//模具切刀
fbMouldCam(
	Reset:=stSysState.bReset , 
	bCamInExecute:=stMouldCam.bCamInExecute , 
	bCreatTable:=stMouldCam.bCreatTable , 
	iTable:=TableNo.Mould , 
	iTableSel:= , 
	fEnterPos:=arrAxisPar[AxisNo.Mould].arrTargetPoint[2] , 
	fLeavePos:=arrAxisPar[AxisNo.Mould].arrTargetPoint[1] , 
	fMainPos:=ProductPar.parPublic.fMainPos , 
	axisSlave:=arrAxis[AxisNo.Mould] , 
	axisMaster:=arrAxis[VirAxisNo.VirMain] , 
	bCreatTableDone=>stMouldCam.bCreatTableDone , 
	bCreatTableError=>stMouldCam.bCreatTableError , 
	bError=>stMouldCam.bError , 
	bReady=>stMouldCam.bReady , 
	bInSync=>stMouldCam.bInSync );
	
//裁切切刀
fbCuterCam(
	Reset:=stSysState.bReset , 
	bCamInExecute:=stCuterCam.bCamInExecute , 
	bCreatTable:=stCuterCam.bCreatTable , 
	iTable:=TableNo.Cuter , 
	iTableSel:= ,
	fEnterPos:=arrAxisPar[AxisNo.Cuter].arrTargetPoint[2] , //裁切切入点角度
	fLeavePos:=arrAxisPar[AxisNo.Cuter].arrTargetPoint[1] , //裁切切尽点角度
	fMainPos:=ProductPar.parPublic.fMainPos , 
	axisSlave:=arrAxis[AxisNo.Cuter] , 
	axisMaster:=arrAxis[VirAxisNo.VirMain] , 
	bCreatTableDone=>stCuterCam.bCreatTableDone , 
	bCreatTableError=>stCuterCam.bCreatTableError , 
	bError=>stCuterCam.bError , 
	bReady=>stCuterCam.bReady , 
	bInSync=>stCuterCam.bInSync );

//CCD压片升降
fbCCDPressCam(
	Reset:=stSysState.bReset , 
	bCamInExecute:=stCCDPressCam.bCamInExecute , 
	bCreatTable:=stCCDPressCam.bCreatTable , 
	iTable:=TableNo.CCDPress , 
	fMainPos:=ProductPar.parPublic.fMainPos , 
	fPressPos:=arrAxisPar[AxisNo.CCDPressPush].arrTargetPoint[2]  , 
	fLeavePos:=arrAxisPar[AxisNo.CCDPressPush].arrTargetPoint[1] , 
	axisSlave:=arrAxis[AxisNo.CCDPressPush]  , 
	axisMaster:=arrAxis[VirAxisNo.VirMain]  , 
	bCreatTableDone=>stCCDPressCam.bCreatTableDone , 
	bCreatTableError=>stCCDPressCam.bCreatTableError , 
	bError=>stCCDPressCam.bError , 
	bReady=>stCCDPressCam.bReady , 
	bInSync=>stCCDPressCam.bInSync );
	
//皮带虚轴
fbVirBeltCam(
	Reset:=stSysState.bReset , 
	bCamInExecute:=stVirBeltCam.bCamInExecute , 
	bCreatTable:=stVirBeltCam.bCreatTable , 
	iTable:=TableNo.VirBelt , 
	fMainPos:=ProductPar.parPublic.fMainPos , 
	fBeltSpacePos:=PolePar.fBeltSpacePos , 
	axisSlave:=arrAxis[VirAxisNo.VirBelt]  , 
	axisMaster:=arrAxis[VirAxisNo.VirMain] , 
	bCreatTableDone=>stVirBeltCam.bCreatTableDone , 
	bCreatTableError=>stVirBeltCam.bCreatTableError , 
	bError=>stVirBeltCam.bError , 
	bReady=>stVirBeltCam.bReady , 
	bInSync=>stVirBeltCam.bInSync );
(*	
//NG踢料
fbNGPushCam(
	Reset:=stSysState.bReset , 
	bCamInExecute:=stNGPushCam.bCamInExecute , 
	bCreatTable:=stNGPushCam.bCreatTable , 
	iTable:=TableNo.NgPush , 
	iTableSel:= , 
	fEnterPos:=arrAxisPar[AxisNo.NGPush2].arrTargetPoint[2] , //NG打料预踢角度 , 
	fLeavePos:=arrAxisPar[AxisNo.NGPush2].arrTargetPoint[1] , //NG打料踢后角度 , 
	fMainPos:=ProductPar.parPublic.fMainPos , 
	axisSlave:=arrAxis[AxisNo.NGPush2] , 
	axisMaster:=arrAxis[VirAxisNo.VirMain] , 
	bCreatTableDone=>stNGPushCam.bCreatTableDone , 
	bCreatTableError=>stNGPushCam.bCreatTableError , 
	bError=>stNGPushCam.bError , 
	bReady=>stNGPushCam.bReady , 
	bInSync=>stNGPushCam.bInSync );
	*)
END_ACTION

ACTION F12TensionCall:


	fbPoleBufferTen.bTensionOK:=stUwindTen.bTensionOK;
	
	fbPoleBufferTen(
	bReset:=                               stSysState.bReset , 
	fAuxDriverDiameter:=            PolePar.Machine.fAuxDriverInDiameter ,  
	fDDRDiameter:=                    PolePar.Machine.fMQDriverDiameter ,  
	fPoleWith:=                           PolePar.fPoleWidth , 
    fCompensation:=                   fPoleBufferCompensation , 
    fDanceBlancePos:=                arrAxisPar[AxisNo.BuffeLine].arrTargetPoint[1] ,  
   	bPositiveLimit:=                     arrAxisCtrl[AxisNo.BuffeLine].Io.biPosLimit   , 
	bNegativeLimit:=                   arrAxisCtrl[AxisNo.BuffeLine].Io.biNegLimit      , 
	bTensionOK:=                       fbPoleBufferTen.bTensionOK     , 
	fMainVel:=                            PolePar.iMainVel         , 
	bReady=>                            stBufferTen.bReady , 
	bError=>                              stBufferTen.bError , 
	bInSync=>                            stBufferTen.bInSync, 
	VirMain:=                             arrAxis[VirAxisNo.VirMain], 
	//AuxDriver:=                          arrAxis[AxisNo.DriverAux] ,
	DDRDriver:=                         arrAxis[AxisNo.DriverDDR]  ,
	VirDriver:=                           arrAxis[VirAxisNo.VirDriver]  ,
	BufferLine:=                         arrAxis[AxisNo.BuffeLine] ,  
	bTenExecute:=                     stBufferTen.bExecute   );
	
	//放卷张力
PolePar.MQ.TenCcw_WindL:=PolePar.MQ.TenCcw_WindR:=FALSE;
	fbUwindTen(
		bReset:=stSysState.bReset , 
		bCcwL:=PolePar.MQ.TenCcw_WindL, //左放卷方向
		bCcwR:=PolePar.MQ.TenCcw_WindR,//右放卷方向
		bWindSel:=PolePar.MQ.bWindSelect, //左右卷选择
		fDiaMin:=250,//最小卷径		
		fDiaMax:=800,//最大卷径
		//fDanserDegree:=arrAxisCtrl[AxisNo.PoleTension].Status.fActPos , 
		fActTorque:= SEL(iPartSelect=1   , iActDriveTorque[2],    iActDriveTorque[1] )    , 
		fSetTorque:= SEL(iPartSelect=1   , iTargetTorque[2],       iTargetTorque[1] )      , 
		PidSwitch:=PolePar.MQ.WindPidSwitch ,
		bTenExecute:=stUwindTen.bTenExecute , 
		bStudyExecute:=stUwindTen.bStudyExecute AND stUwindTen.fStudyDiameter>0, 
		fStudyDiameter:=stUwindTen.fStudyDiameter , 
		fDriveDiameter:=PolePar.Machine.fMQDriverDiameter, 
		fPoleWith:=PolePar.fPoleWidth , 
		fCompensation:= , 
		fDancerMinPos:=PolePar.MQ.AuxDriverTenMinPos,//摆杆最小角度
		fDancerMaxPos:=PolePar.MQ.AuxDriverTenMaxPos,//摆杆最大角度
		fDanceBlancePos:=PolePar.MQ.AuxDriverTenBlancePos , //摆杆平衡角度
		fDanserDegree:=stAuxDriverTen.fDanserDegree , //摆杆实时角度
		//fDancerMinPos:=PolePar.MQ.WindTenMinPos , 
		//fDancerMaxPos:=PolePar.MQ.WindTenMaxPos , 
		//fDanceBlancePos:=PolePar.MQ.WindTenBlancePos , 
		bReady=>stUwindTen.bReady , 
		bTensionOK=>stUwindTen.bTensionOK , 
		bError=>stUwindTen.bError , 
		fWindDiameterTemp=>stUwindTen.fWindDiameter,
		VirMain:=arrAxis[VirAxisNo.VirMain] , 
		Master:=arrAxis[VirAxisNo.VirDriver] , 
		SlaveL:=arrAxis[AxisNo.UnWind_L], 
		SlaveR:=arrAxis[AxisNo.UnWind_R], 
		Driver:=arrAxis[AxisNo.DriverDDR] , 
		TimerAxis:=arrAxis[NameNo.VirTimeWind] , 
		TensionAxis:=arrAxis[AxisNo.PoleTension] , 
		Table:=PolePar.MQ.WindTenTable ,
		AxisNoBuffeLine :=AxisNo.BuffeLine);
	

		
		
(*
//左放卷张力

fbUwindLTen(
	bReset:=stSysState.bReset , 
	bCcw:=PolePar.MQ.TenCcw_WindL , 
	fDanserDegree:=stUwindLTen.fDanserDegree , 
	//fWindDiameter:=stUwindLTen.fWindDiameter  , 
	fActTorque:= SEL(iPartSelect=1   , iActDriveTorque[2],    iActDriveTorque[1] )    , 
	fSetTorque:= SEL(iPartSelect=1   , iTargetTorque[2],       iTargetTorque[1] )      , 
	PidSwitch:=TRUE , //PolePar.MQ.WindPidSwitch
	bTenExecute:=stUwindLTen.bTenExecute , 
	bStudyExecute:=stUwindLTen.bStudyExecute , 
	fStudyDiameter:=stUwindLTen.fStudyDiameter , 
	fDriveDiameter:=PolePar.Machine.fAuxDriverInDiameter , 
	fPoleWith:=PolePar.fPoleWidth , 
	fCompensation:= , 
	fDancerMinPos:=PolePar.MQ.WindTenMinPos , 
	fDancerMaxPos:=PolePar.MQ.WindTenMaxPos , 
	fDanceBlancePos:=PolePar.MQ.WindTenBlancePos , 
	bReady=>stUwindLTen.bReady , 
	bTensionOK=>stUwindLTen.bTensionOK , 
	bError=>stUwindLTen.bError , 
	VirMain:=arrAxis[VirAxisNo.VirMain] , 
	Master:=arrAxis[VirAxisNo.VirDriver] , 
	Slave:=arrAxis[AxisNo.UnWind_L] , 
	Driver:=arrAxis[AxisNo.DriverAux] , 
	TimerAxis:=arrAxis[NameNo.VirTimeWind] , 
	TensionAxis:=arrAxis[AxisNo.PoleTension] , 
	Table:=PolePar.MQ.WindTenTable );
	stUwindLTen.fDanserDegree:=arrAxisCtrl[AxisNo.PoleTension].Status.fActPos;
	PolePar.MQ.TenCcw_WindL:=FALSE;
	
	stUwindLTen.fWindDiameter  ;
	fbUwindLTen.fWindDiameter;
	fbUwindLTen.fDiameterCalculate;
	fbUwindLTen.fWindDiameterTemp;
	
//右放卷张力
fbUwindRTen(	
	bReset:=stSysState.bReset , 
	bCcw:=PolePar.MQ.TenCcw_WindR , 
	fDanserDegree:=stUwindRTen.fDanserDegree , 
	//fWindDiameter:=stUwindRTen.fWindDiameter , 
	fActTorque:= SEL(iPartSelect=1   , iActDriveTorque[2],    iActDriveTorque[1] )    , 
	fSetTorque:= SEL(iPartSelect=1   , iTargetTorque[2],       iTargetTorque[1] )      , 
	PidSwitch:=TRUE, //PolePar.MQ.WindPidSwitch 
	bTenExecute:=stUwindRTen.bTenExecute , 
	bStudyExecute:=stUwindRTen.bStudyExecute , 
	fStudyDiameter:=stUwindRTen.fStudyDiameter , 
	fDriveDiameter:=PolePar.Machine.fAuxDriverInDiameter , 
	fPoleWith:=PolePar.fPoleWidth , 
	fCompensation:= ,
	fDancerMinPos:=PolePar.MQ.WindTenMinPos , 
	fDancerMaxPos:=PolePar.MQ.WindTenMaxPos , 
	fDanceBlancePos:=PolePar.MQ.WindTenBlancePos , 
	bReady=>stUwindRTen.bReady , 
	bTensionOK=>stUwindRTen.bTensionOK , 
	bError=>stUwindRTen.bError , 
	VirMain:=arrAxis[VirAxisNo.VirMain] , 
	Master:=arrAxis[VirAxisNo.VirDriver] , 
	Slave:=arrAxis[AxisNo.UnWind_R]  , 
	Driver:=arrAxis[AxisNo.DriverAux] , 
	TimerAxis:=arrAxis[NameNo.VirTimeWind], 
	TensionAxis:=arrAxis[AxisNo.PoleTension] , 
	Table:=PolePar.MQ.WindTenTable );
	
	
	
	stUwindRTen.fDanserDegree:=arrAxisCtrl[AxisNo.PoleTension].Status.fActPos;
	PolePar.MQ.TenCcw_WindR:=FALSE;
	
	stUwindRTen.fWindDiameter  ;
	fbUwindRTen.fWindDiameter;
	fbUwindRTen.fDiameterCalculate;
	fbUwindRTen.fWindDiameterTemp;
*)	
//辅驱张力
stAuxDriverTen.fWindDiameter:=stAuxDriverTen.fStudyDiameter:=PolePar.Machine.fAuxDriverInDiameter;
PolePar.MQ.TenCcw_AuxDriver:=FALSE;
fbAuxDriverTen(
	bReset:=stSysState.bReset , 
	bCcw:=PolePar.MQ.TenCcw_AuxDriver , 
	fDanserDegree:=stAuxDriverTen.fDanserDegree , 
	fWindDiameter:=stAuxDriverTen.fWindDiameter , 
	PidSwitch:=FALSE , //PolePar.MQ.AuxDriverPidSwitch
	bTenExecute:=stAuxDriverTen.bTenExecute , 
	bStudyExecute:=FALSE, //stAuxDriverTen.bStudyExecute
	fStudyDiameter:=stAuxDriverTen.fStudyDiameter , 
	fPoleWith:=PolePar.fPoleWidth , 
	fCompensation:= , 
	fDancerMinPos:=PolePar.MQ.AuxDriverTenMinPos , 
	fDancerMaxPos:=PolePar.MQ.AuxDriverTenMaxPos , 
	fDanceBlancePos:=PolePar.MQ.AuxDriverTenBlancePos , 
	bReady=>stAuxDriverTen.bReady , 
	bTensionOK=>stAuxDriverTen.bTensionOK , 
	bError=>stAuxDriverTen.bError , 
	VirMain:=arrAxis[VirAxisNo.VirMain] , 
	Master:=arrAxis[VirAxisNo.VirDriver] , 
	Slave:=arrAxis[AxisNo.DriverAux] , 
	TimerAxis:=arrAxis[NameNo.VirTimeWind] , 
	Table:=PolePar.MQ.AuxDriverTenTable );
END_ACTION

ACTION F13ClearBelt:
//一键皮带清料
rtClearBelt[1](CLK:=SysPart.hmiClearBelt , Q=> );
rtClearBelt[2](CLK:= , Q=> );
rtClearBelt[3](CLK:= , Q=> );
rtClearBelt[4](CLK:= , Q=> );
rtClearBelt[5](CLK:= , Q=> );
tonClearBelt[1](In:=,PT:=T#200MS);
tonClearBelt[2](In:=,PT:=T#200MS);
tonClearBelt[3](In:=,PT:=T#200MS);
tonClearBelt[4](In:=,PT:=T#200MS);	
tonClearBelt[5](In:=,PT:=T#200MS);	
tonClearBelt[6](In:=,PT:=T#200MS);	
tonClearBelt[7](In:=,PT:=T#200MS);
tonClearBelt[8](In:=,PT:=T#200MS);
tonClearBelt[9](In:=,PT:=T#200MS);
tonClearBelt[10](In:=,PT:=T#200MS);
IF rtClearBelt[1].Q THEN
	iClearBeltStep:=88;//皮带清料触发
END_IF;

CASE iClearBeltStep OF
///////////////////////////////////////////////////////////凸轮耦合/////////////////////////////////////////////////////
88://有关气缸动作
	arrCyCtrl[CYNo.NGRevBeltTension].Cmd.bON:=TRUE;
	arrCyCtrl[CYNo.NGRevBeltUpDown].Cmd.bON:=TRUE;
	arrCyCtrl[CYNo.DustRevBeltUpDown].Cmd.bON:=TRUE;
	IF	arrCyCtrl[CyNo.NGRevBeltUpDown].Status.ONState AND arrCyCtrl[CYNo.DustRevBeltUpDown].Status.ONState THEN
		iClearBeltStep:=90;//		
	END_IF
	
90://凸轮/张力解耦
	bMethodTenBufferDisEnable:=TRUE;
	bMethodCamDisEnable:=TRUE;
	iClearBeltStep:=100;//	
	
100://判断是否解耦完成
	IF NOT bMethodTenBufferDisEnable AND NOT bMethodCamDisEnable THEN
		iClearBeltStep:=110;
	END_IF
110://主轴清0
	IF arrAxisCtrl[VirAxisNo.VirMain].Status.fModuloActPos<>0 THEN
		arrAxisCtrl[VirAxisNo.VirMain].Cmd.fSetPos:=arrAxisCtrl[VirAxisNo.VirMain].Status.fActPos-arrAxisCtrl[VirAxisNo.VirMain].Status.fModuloActPos+360;
		arrAxisCtrl[VirAxisNo.VirMain].Cmd.bSetPos:=TRUE;
	END_IF
	iClearBeltStep:=120;
120://皮带虚轴耦合
	IF NOT stVirBeltCam.bInSync THEN
		stVirBeltCam.bCamInExecute:=TRUE;
	ELSE
		iClearBeltStep:=130;
	END_IF	
130://皮带齿合
	IF NOT stCuterBeltGear.bInGear THEN
		stCuterBeltGear.bEnable:=TRUE;
	END_IF	
	IF NOT stNGReverseBeltGear.bInGear THEN
		stNGReverseBeltGear.bEnable:=TRUE;
	END_IF		
	IF NOT stDedustBeltGear.bInGear THEN
		stDedustBeltGear.bEnable:=TRUE;
	END_IF
	IF NOT stDedustReverseBeltGear.bInGear THEN
		stDedustReverseBeltGear.bEnable:=TRUE;
	END_IF

	IF NOT stSubBelt1Gear.bInGear THEN
		stSubBelt1Gear.bEnable:=TRUE;
	END_IF

	IF NOT stSubBelt2Gear.bInGear THEN
		bSubBelt2fratio:=TRUE;
		stSubBelt2Gear.bEnable:=TRUE;
	END_IF	
	
	IF NOT stSubBelt3Gear.bInGear THEN
		bSubBelt3fratio:=TRUE;
		stSubBelt3Gear.bEnable:=TRUE;
	END_IF		

	IF stCuterBeltGear.bInGear AND stNGReverseBeltGear.bInGear AND stDedustBeltGear.bInGear AND stDedustReverseBeltGear.bInGear AND 
	     stSubBelt1Gear.bInGear AND  stSubBelt2Gear.bInGear AND  stSubBelt3Gear.bInGear THEN
    	iClearBeltStep:=140;		
	END_IF
140://主轴运动40个周期
	arrAxisCtrl[VirAxisNo.VirMain].Cmd.bDynamitcsParSel:=1;
	arrAxisCtrl[VirAxisNo.VirMain].Cmd.fPositon_of_Abs:=arrAxisCtrl[VirAxisNo.VirMain].Status.fActPos-arrAxisCtrl[VirAxisNo.VirMain].Status.fModuloActPos+40*360;
	arrAxisPar[VirAxisNo.VirMain].fVelocity_of_Abs:=PolePar.iMainVel*6;
	arrAxisCtrl[VirAxisNo.VirMain].Cmd.bMoveAbs:=TRUE;
	IF arrAxisCtrl[VirAxisNo.VirMain].Status.Moving THEN
		iClearBeltStep:=150;
	END_IF
150://判断主轴运动完成
	IF arrAxisCtrl[VirAxisNo.VirMain].Status.NoMoving AND NOT arrAxisCtrl[VirAxisNo.VirMain].Cmd.bMoveAbs THEN
		iClearBeltStep:=160;
	END_IF
160://清除皮带记忆
	MEMSET(ADR(BeltData),0,SIZEOF(BeltData));
	iClearBeltStep:=170;
170://
	SysPart.hmiClearBelt:=FALSE;
	iClearBeltStep:=666;

END_CASE
END_ACTION

ACTION Product:

//切刀计数
rtCount2(CLK:=arrAxisCtrl[VirAxisNo.VirMain].Status.fModuloActPos>=10 AND arrAxisCtrl[VirAxisNo.VirMain].Status.fModuloActPos<=100);
IF rtCount2.Q THEN
	Production.OutFlag1:=TRUE;//产能计数
END_IF

////////////////////////////////////////////////////////////////NG剔废////////// NG分类 //////////////////////////////////////////////////////
ProductPar.iModeEN.bNG1PushEN:=ProductPar.iModeEN.bNG2PushEN;
CASE iNGStep OF 
10://判断NG1&NG2是否动作 主轴静止或运行中
	IF (  NOT ProductPar.iModeEN.bEmptyRunEN AND NOT ProductPar.iModeEN.bSizeCCDEN AND BeltData[BeltNo.NGBox1+2].fPoleNGSizeNo<>30 ) THEN//BeltData[BeltNo.NGBox].iPanoramaNG<>1
		 iNGStep:=200;
	ELSIF  BeltData[BeltNo.NGBox1+2].fPoleNGSacnNo<>30   AND NOT ProductPar.iModeEN.bLineScanCCDEN  THEN //XianSaong_Up[2]<>30 OR XianSaong_Down[0]<>30  
		iNGStep:=300;
	ELSIF  BeltData[BeltNo.NGBox1+2].bYellowMark    OR  BeltData[BeltNo.NGBox1+2].bBlueMark  THEN//黄标
		iNGStep:=300;
	ELSE
		nInt[3]:=0;
		arrCyCtrl[EvNo.	NGPushInsideAir	].Cmd.bON:=FALSE;//踢NG料打开
		arrCyCtrl[EvNo.	NGPushInsideAir	].Cmd.bOFF:=TRUE;//踢NG料关闭		
		arrCyCtrl[EVNo.NGPushInsideVacuo].Cmd.bON:=TRUE;//踢NG料真空打开
		arrCyCtrl[EVNo.NGPushInsideVacuo].Cmd.bOFF:=FALSE;//踢NG料真空关闭		
		iNGStep:=666;
	END_IF

200:
	IF  NOT ProductPar.iModeEN.bEmptyRunEN   THEN//AND NOT  ProductPar.iModeEN.bP2PartEN
			IF REAL_TO_INT(BeltData[BeltNo.NGBox1+2].fPoleNGSizeNo)=1 THEN
				Production.NGFlag[49]:=TRUE;//尺寸总不良
				Production.NGFlag[1]:=TRUE;//极片长度不良
			ELSIF REAL_TO_INT(BeltData[BeltNo.NGBox1+2].fPoleNGSizeNo)=2 THEN
				Production.NGFlag[49]:=TRUE;//尺寸总不良
				Production.NGFlag[2]:=TRUE;//极片CIL宽度不良
			ELSIF REAL_TO_INT(BeltData[BeltNo.NGBox1+2].fPoleNGSizeNo)=3 THEN
				Production.NGFlag[49]:=TRUE;//尺寸总不良
				Production.NGFlag[3]:=TRUE;//极片宽度不良标志位
			ELSIF REAL_TO_INT(BeltData[BeltNo.NGBox1+2].fPoleNGSizeNo)=4 THEN
				Production.NGFlag[49]:=TRUE;//尺寸总不良
				Production.NGFlag[4]:=TRUE;//极耳宽度不良
			ELSIF REAL_TO_INT(BeltData[BeltNo.NGBox1+2].fPoleNGSizeNo)=5 THEN
				Production.NGFlag[49]:=TRUE;//尺寸总不良
				Production.NGFlag[5]:=TRUE;//极耳高度不良
			ELSIF REAL_TO_INT(BeltData[BeltNo.NGBox1+2].fPoleNGSizeNo)=6 THEN
				Production.NGFlag[49]:=TRUE;//尺寸总不良
				Production.NGFlag[6]:=TRUE;//极耳侧边距不良
			ELSIF REAL_TO_INT(BeltData[BeltNo.NGBox1+2].fPoleNGSizeNo)=7 THEN
				Production.NGFlag[49]:=TRUE;//尺寸总不良
				Production.NGFlag[7]:=TRUE;//极耳面积不良
			ELSIF REAL_TO_INT(BeltData[BeltNo.NGBox1+2].fPoleNGSizeNo)=8 THEN
				Production.NGFlag[49]:=TRUE;//尺寸总不良
				Production.NGFlag[8]:=TRUE;//圆角深度不良
			ELSIF REAL_TO_INT(BeltData[BeltNo.NGBox1+2].fPoleNGSizeNo)=9 THEN
				Production.NGFlag[49]:=TRUE;//尺寸总不良
				Production.NGFlag[9]:=TRUE;//极耳边缘角度不良
			ELSIF REAL_TO_INT(BeltData[BeltNo.NGBox1+2].fPoleNGSizeNo)=10 THEN
				Production.NGFlag[49]:=TRUE;//尺寸总不良
				Production.NGFlag[10]:=TRUE;//圆角宽度不良
			ELSIF REAL_TO_INT(BeltData[BeltNo.NGBox1+2].fPoleNGSizeNo)=11 THEN
				Production.NGFlag[49]:=TRUE;//尺寸总不良
				Production.NGFlag[11]:=TRUE;//圆角轮廓不良	
			ELSIF REAL_TO_INT(BeltData[BeltNo.NGBox1+2].fPoleNGSizeNo)=12 THEN
				Production.NGFlag[49]:=TRUE;//尺寸总不良
				Production.NGFlag[12]:=TRUE;//圆角面积不良		
			ELSIF REAL_TO_INT(BeltData[BeltNo.NGBox1+2].fPoleNGSizeNo)=13 THEN
				Production.NGFlag[49]:=TRUE;//尺寸总不良
				Production.NGFlag[13]:=TRUE;//圆角余料不良		
			ELSIF (BeltData[BeltNo.NGBox1+2].fPoleNGSizeNo<>1 AND BeltData[BeltNo.NGBox1+2].fPoleNGSizeNo<>2 AND BeltData[BeltNo.NGBox1+2].fPoleNGSizeNo<>3
				AND BeltData[BeltNo.NGBox1+2].fPoleNGSizeNo<>4 AND BeltData[BeltNo.NGBox1+2].fPoleNGSizeNo<>5 AND BeltData[BeltNo.NGBox1+2].fPoleNGSizeNo<>6
				 AND BeltData[BeltNo.NGBox1+2].fPoleNGSizeNo<>7  AND BeltData[BeltNo.NGBox1+2].fPoleNGSizeNo<>8  AND BeltData[BeltNo.NGBox1+2].fPoleNGSizeNo<>9
				 AND BeltData[BeltNo.NGBox1+2].fPoleNGSizeNo<>11  AND BeltData[BeltNo.NGBox1+2].fPoleNGSizeNo<>12  AND BeltData[BeltNo.NGBox1+2].fPoleNGSizeNo<>13
				) OR  BeltData[BeltNo.NGBox1+2].fPoleNGSizeNo=33  THEN  //尺寸检测其他不良 ,,,CCD超时
				Production.NGFlag[49]:=TRUE;//尺寸检测其他不良 ,,,CCD超时
				Production.NGFlag[14]:=TRUE;
			END_IF
	END_IF
		FOR i:=1 TO 20 DO
			IF i<20 THEN
				XianSaong[21-i]:=XianSaong[20-i];
				XianSaong1[21-i]:=XianSaong1[20-i];
			ELSE
				XianSaong[1]:=BeltData[BeltNo.NGBox1].iPanoramaNG;
				XianSaong1[1]:=REAL_TO_INT(BeltData[BeltNo.NGBox1].fPoleNGSizeNo);
			END_IF
		END_FOR
		iNGStep:=400;
300:
	 IF NOT ProductPar.iModeEN.bEmptyRunEN  THEN//AND NOT  ProductPar.iModeEN.bP2PartEN
			IF BeltData[BeltNo.NGBox1+2].fPoleNGSacnNo=1 THEN
				Production.NGFlag[48]:=TRUE;//线扫总不良
				Production.NGFlag[21]:=TRUE;//抓边失败
			ELSIF BeltData[BeltNo.NGBox1+2].fPoleNGSacnNo=2 THEN
				Production.NGFlag[48]:=TRUE;//线扫总不良
				Production.NGFlag[22]:=TRUE;//直边不良标志位
			ELSIF BeltData[BeltNo.NGBox1+2].fPoleNGSacnNo=3 THEN
				Production.NGFlag[48]:=TRUE;//线扫总不良
				Production.NGFlag[23]:=TRUE;//极片缺失
			ELSIF BeltData[BeltNo.NGBox1+2].fPoleNGSacnNo=4 THEN
				Production.NGFlag[48]:=TRUE;//线扫总不良
				Production.NGFlag[24]:=TRUE;//接带
			ELSIF BeltData[BeltNo.NGBox1+2].fPoleNGSacnNo=5 THEN
				Production.NGFlag[48]:=TRUE;//线扫总不良
				Production.NGFlag[25]:=TRUE;//线扫黄标
			ELSIF BeltData[BeltNo.NGBox1+2].fPoleNGSacnNo=6 THEN
				Production.NGFlag[48]:=TRUE;//线扫总不良
				Production.NGFlag[26]:=TRUE;//漏金属
			ELSIF BeltData[BeltNo.NGBox1+2].fPoleNGSacnNo=7 THEN
				Production.NGFlag[48]:=TRUE;//线扫总不良
				Production.NGFlag[27]:=TRUE;//气泡
			ELSIF BeltData[BeltNo.NGBox1+2].fPoleNGSacnNo=8 THEN
				Production.NGFlag[48]:=TRUE;//线扫总不良
				Production.NGFlag[28]:=TRUE;//暗条痕
			ELSIF BeltData[BeltNo.NGBox1+2].fPoleNGSacnNo=9 THEN
				Production.NGFlag[48]:=TRUE;//线扫总不良
				Production.NGFlag[29]:=TRUE;//亮条痕
			ELSIF BeltData[BeltNo.NGBox1+2].fPoleNGSacnNo=10 THEN
				Production.NGFlag[48]:=TRUE;//线扫总不良
				Production.NGFlag[30]:=TRUE;//破损
			ELSIF BeltData[BeltNo.NGBox1+2].fPoleNGSacnNo=11 THEN
				Production.NGFlag[48]:=TRUE;//线扫总不良
				Production.NGFlag[31]:=TRUE;//碎屑
			ELSIF BeltData[BeltNo.NGBox1+2].fPoleNGSacnNo=12 THEN
				Production.NGFlag[48]:=TRUE;//线扫总不良
				Production.NGFlag[33]:=TRUE;//脱碳
			ELSIF BeltData[BeltNo.NGBox1+2].fPoleNGSacnNo=29 THEN
				Production.NGFlag[48]:=TRUE;//线扫总不良
				Production.NGFlag[34]:=TRUE;//其他
			ELSIF BeltData[BeltNo.NGBox1+2].fPoleNGSacnNo=33 THEN
				Production.NGFlag[48]:=TRUE;//线扫总不良
				Production.NGFlag[32]:=TRUE;//通讯超时
(*			ELSIF BeltData[BeltNo.NGBox1+2].bYellowMark  THEN
				//Production.NGFlag[48]:=TRUE;//线扫总不良
				Production.NGFlag[33]:=TRUE;//感应器黄标*)
			END_IF
	END_IF
		iNGStep:=400;
400:
	arrCyCtrl[EvNo.	NGPushInsideAir	].Cmd.bON:=TRUE;//踢NG料破真空打开
	arrCyCtrl[EvNo.	NGPushInsideAir	].Cmd.bOFF:=FALSE;//踢NG料破真空关闭
	arrCyCtrl[EVNo.NGPushInsideVacuo].Cmd.bON:=FALSE;//踢NG料真空打开
	arrCyCtrl[EVNo.NGPushInsideVacuo].Cmd.bOFF:=TRUE;//踢NG料真空关闭
	BeltData[BeltNo.NGBox1+2].bHavePole:=FALSE;	
	BeltData[BeltNo.NGBox1+2].stPoleNo:='';
	nInt[3]:=1;		
	//BeltData[BeltNo.NGBox1].bHavePole:=FALSE;
	FOR i:=1 TO 50 DO//NG类型标志位复位
		Production.NGFlag[i]:=FALSE;
    	END_FOR
	iNGStep:=666;
END_CASE

IF iNGStep=300 THEN
	IF BeltData[BeltNo.NGBox1+1].bBlueMark OR BeltData[BeltNo.NGBox1+2].bBlueMark OR BeltData[BeltNo.NGBox1+3].bBlueMark THEN
		iNGState:=1;//接带踢废
	ELSIF BeltData[BeltNo.NGBox1+2].bYellowMark THEN
		IF BeltData[BeltNo.NGBox1+1].bYellowMark THEN
			iNGState:=2;//黄标跳切踢废
		ELSIF NOT BeltData[BeltNo.NGBox1+3].bYellowMark THEN
			iNGState:=3;//黄标单张踢废
		END_IF
	ELSIF BeltData[BeltNo.NGBox1+2].fPoleNGSacnNo=4 THEN
		iNGState:=4;//线扫接带
	ELSIF BeltData[BeltNo.NGBox1+2].fPoleNGSacnNo=5 THEN
		iNGState:=5;//线扫黄标
	END_IF
END_IF

aFB_ProductionDataLocal(
	NowTimeData:=System.StTime, (*当前系统时间*)
	OutFlag1:=Production.OutFlag1, (*产量计数标志1*)
	OutFlag2:=Production.OutFlag2, (*产量计数标志1*)
	NGFlag:=Production.NGFlag ,(*NG1计数标志*)(*扫码NG*)
	RunFlag:=stSysState.iMode=1,(*运行标志*)
	WaitFlag:=stSysState.iMode<>1 AND NOT stSysState.Alarming ,(*待料标志*)
	AlarmFlag:=stSysState.Alarming, (*故障标志*)
	DelDataAMBtn:= Production.HMI_DelDataAMBtn,(*白班数据清除按钮*)//HMI_DayCountZero
	DelDataPMBtn:= Production.HMI_DelDataPMBtn,(*夜班数据清除按钮*)//HMI_NightCountZero
	NowOutTotal=>Production.HMI_TotalCount ,(*当前班次加工总数*)
	NowRate=> Production.HMI_Qualified,(*当前班次良率*)
	NGClearAMBtn:=Production.HMI_NGClearAMBtn,//白班NG类型计数清零
	NGClearPMBtn:=Production.HMI_NGClearPMBtn,//夜班NG类型计数清零
	NowDay:= Production.SaveNowDay,(*数据移位时所保存当前日*)
	NowMonth:=Production.SaveNowMonth ,(*数据移位时所保存当前月*)
	DayHistory:= Production.DayReadDayHistory, (*历史日*)
	MonthHistory:= Production.DayReadMonthHistory,(*历史月*)
	TodayTotal:=Production.HMI_TodayTotal ,(*当天24H生产总数*)
	TodayOK:=Production.HMI_TodayOK , (*当天24H生产OK总数*)
	TodayNG:=Production.HMI_TodayNG , (*当天24H生产NG总数*)
	TodayTotal_AM:= Production.DayCountTotal,(*当天白班生产总数*)
	TodayTotal_PM:=Production.NightCountTotal,(*当天夜班生产总数*)
	TodayRate_AM:= Production.HMI_DayQualified,(*当天白班良率*)
	TodayRate_PM:=Production.HMI_NightQualified ,(*当天夜班良率*)
	OEE=> Production.HMI_OEE,//设备稼动率/稼动率
	TodayOK_AM:=Production.HMI_DayOkCount ,(*当天白班生产OK总数*)
	TodayOK_PM:= Production.HMI_NightOkCount,(*当天夜班生产OK总数*)
	TodayNG_AM:=Production.HMI_DayNgCount ,(*当天白班生产NG总数*)
	TodayNG_PM:=Production.HMI_NightNgCount , (*当天夜班生产NG总数*)
	TodayHour_AM:= Production.HourTimeDayCount,(*当天白班每小时产量ARRAY[8..19 ]*)
	TodayHour_PM:=Production.HourTimeNightCount ,(*当天夜班每小时产量ARRAY[0..23]*)
	TodayNGClass_AM:=Production.NgPerHourDayCount , (*当天白班各类NG数量ARRAY[1..30 ]*)
	TodayNGClass_PM:= Production.NgPerHourNightCount,(*当天夜班各类NG数量ARRAY[1..30 ]*)
	TodayRun_AM:= Production.DayRunTimeTotal,(*当天白班总运行时间合计/分*)
	TodayRun_PM:= Production.NightRunTimeTotal,(*当天夜班总运行时间合计/分*)
	TodayWait_AM:=Production.DayWaitTimeTotal , (*当天白班总待料时间合计/分*)
	TodayWait_PM:=Production.NightWaitTimeTotal , (*当天夜班总待料时间合计/分*)
	TodayAlarm_AM:=Production.DayAlarmTimeTotal ,(*当天白班总报警时间合计/分*)
	TodayAlarm_PM:=Production.NightAlarmTimeTotal, (*当天夜班总报警时间合计/分*)
	
	TodayRun_AMH:=Production.DayRunTime_min,(*当天白班每小时运行时间合计/分*)
	TodayRun_PMH:=Production.NightRunTime_min,(*当天夜班每小时运行时间合计/分*)
	TodayWait_AMH:=Production.DayWaitTime_min,(*当天白班每小时待料时间合计/分*)
	TodayWait_PMH:=Production.NightWaitTime_min,(*当天夜班每小时待料时间合计/分*)
	TodayAlarm_AMH:=Production.DayAlmTime_min,(*当天白班每小时报警时间合计/分*)
	TodayAlarm_PMH:=Production.NightAlmTime_min,(*当天夜班每小时报警时间合计/分*)
	
	HistoryRun_AMH:=Production.HisDayRunTime_min,(*历史每天白班每小时运行时间合计ARRAY[1..7 ]*)
	HistoryRun_PMH:=Production.HisNightRunTime_min,(*历史每天夜班每小时运行时间合计ARRAY[1..7 ]*)
	HistoryWait_AMH:=Production.HisDayWaitTime_min,(*历史每天白班每小时待料时间合计ARRAY[1..7 ]*)
	HistoryWait_PMH:=Production.HisNightWaitTime_min,(*历史每天夜班每小时待料时间合计ARRAY[1..7 ]*)
	HistoryAlarm_AMH:=Production.HisDayAlmTime_min,(*历史每天白班每小时报警时间合计ARRAY[1..7 ]*)
	HistoryAlarm_PMH:=Production.HisNightAlmTime_min,(*历史每天夜班每小时报警时间合计ARRAY[1..7 ]*)
	
	RunCnt_AM:=Production.nDayRunTimeCnt , (*白班运行时间计数*)
	RunCnt_PM:=Production.nNightRunTimeCnt ,(*夜班运行时间计数*)
	WaitCnt_AM:= Production.nDayWaitTimeCnt, (*白班待料时间计数*)
	WaitCnt_PM:=Production.nNightWaitTimeCnt ,(*夜班待料时间计数*)
	AlarmCnt_AM:=Production.nDayAlarmTimeCnt , (*白班报警时间计数*)
	AlarmCnt_PM:= Production.nNightAlarmTimeCnt,(*夜班报警时间计数*)
	
	HistoryTotal:=Production.HMI_HistoryTotal ,(*历史每天24H生产总数ARRAY[1..7 ]*)
	HistoryOK:=Production.HMI_HistoryOK ,(*历史每天24H生产OK总数ARRAY[1..7 ]*)
	HistoryNG:=Production.HMI_HistoryNG , (*历史每天24H生产NG总数ARRAY[1..7 ]*)
	HistoryTotal_AM:=Production.DayCountTotalHistory ,(*历史每天白班生产总数ARRAY[1..7 ]*)
	HistoryTotal_PM:=Production.NightCountTotalHistory ,(*历史每天夜班生产总数ARRAY[1..7 ]*)
	HistoryRate_AM:=Production.HMI_DayQualifiedHistory , (*历史每天白班良率ARRAY[1..7 ]*)
	HistoryRate_PM:=Production.HMI_NightQualifiedHistory,(*历史每天夜班良率ARRAY[1..7 ]*)
	HistoryOK_AM:=Production.HMI_DayOkCountHistory , (*历史每天白班生产OK总数ARRAY[1..7 ]*)
	HistoryOK_PM:=Production.HMI_NightOkCountHistory , (*历史每天夜班生产OK总数ARRAY[1..7 ]*)
	HistoryNG_AM:=Production.HMI_DayNgCountHistory ,(*历史每天白班生产NG总数ARRAY[1..7 ]*)
	HistoryNG_PM:= Production.HMI_NightNgCountHistory,(*历史每天夜班生产NG总数ARRAY[1..7 ]*)
	HistoryHour_AM:=Production.HourTimeDayCountHistory ,(*历史每天白班每小时产量ARRAY[1..7,8..19 ]*)
	HistoryHour_PM:=Production.HourTimeNightCountHistory ,(*历史每天夜班每小时产量ARRAY[1..7,0..23]*)
	HistoryNGClass_AM:= Production.NgPerHourDayCountHistory,(*历史每天白班各类NG数量ARRAY[1..7,1..30 ]*)
	HistoryNGClass_PM:= Production.NgPerHourNightCountHistory,(*历史每天夜班各类NG数量ARRAY[1..7,1..30 ]*)
	HistoryRun_AM:=Production.DayRunTimeTotalHistory , (*历史每天白班总运行时间合计ARRAY[1..7 ]*)
	HistoryRun_PM:= Production.NightRunTimeTotalHistory, (*历史每天夜班总运行时间合计ARRAY[1..7 ]*)
	HistoryWait_AM:= Production.DayWaitTimeTotalHistory,(*历史每天白班总待料时间合计ARRAY[1..7 ]*)
	HistoryWait_PM:= Production.NightWaitTimeTotalHistory, (*历史每天夜班总待料时间合计ARRAY[1..7 ]*)
	HistoryAlarm_AM:= Production.DayAlarmTimeTotalHistory,(*历史每天白班总报警时间合计ARRAY[1..7 ]*)
	HistoryAlarm_PM:= Production.NightAlarmTimeTotalHistory,(*历史每天夜班总报警时间合计ARRAY[1..7 ]*)

	TodayNgHour_Day:=Production.HMINgClassCount_Day,(*白班每种NG类型每小时统计 ,,,NG类型，小时*)
	TodayNgHour_Night:=Production.HMINgClassCount_Night,(*夜班每种NG类型每小时统计 ,,,NG类型，小时*)
	HisTodayNgHour_Day:=Production.HisHMINgClassCount_Day,//l历史白班每小时NG类型统计,,
	HisTodayNgHour_Night:=Production.HisHMINgClassCount_Night,//历史夜班每小时NG类型统计,,
		
	TodayNGQualified:=Production.HMI_TodayNGQualified,//当天白班各种NG类型NG率
	NightNGQualified:=Production.HMI_NightNGQualified,//当天夜班各种NG类型NG率	
	HisTodayNGQualified:=Production.HMI_HisTodayNGQualified,//历史白班各种NG类型NG率
	HisNightNGQualified:=Production.HMI_HisNightNGQualified,//历史夜班各种NG类型NG率
	
	);
END_ACTION

END_FUNCTION_BLOCK

// ---- POUs/BasicFunction/Motion/FB_TailCurl_PID.TcPOU
FUNCTION_BLOCK FB_TailCurl_PID
VAR_INPUT
	ModuloActPos:REAL;//主轴位置；
	sStar:R_TRIG;//固定2个感应器基准值;
	Enable:BOOL;//启动条件
	RestHMI:BOOL;//报警复位
	MasterNo:INT;//主轴号
	SlaveNo:INT;//从轴号
	MasterValue:REAL;//主轴匀速运行时的速度
	//RecDevagree:BOOL;//纠偏许可
	RecDevEqupos1:REAL;//纠偏平传感器1基准值
	RecDevEqupos2:REAL;//纠偏平传感器2基准值
	RecDevValueSet:REAL;//纠偏设定
	RecDevPV1:REAL;//纠偏传感器1实时值
	RecDevPV2:REAL;//纠偏传感器2实时值
	RecDevSpeedCoe:REAL;//纠偏带速度系数
	CWW:BOOL;//纠偏方向选择
	AxisintiPos:REAL;//轴的初始位置
	AxisPos_H:REAL;//轴的纠偏行程上限
	AxisPos_L:REAL;//轴的纠偏行程下限
	bMode:INT;//1=单边纠偏     2=双边纠偏
	iMainVel: UINT;
END_VAR
VAR_OUTPUT
	//RecDevSpeed:REAL;//纠偏速度
	bError:BOOL;
	JZError:ARRAY [0..10] OF BOOL;//双纠偏传感器错误；
	bRecOK: BOOL;
	bReady: BOOL;
END_VAR
VAR
	// 执行延时2S
	TON1: TON;
	// 轴纠偏上限
	AxisRecDevPos_H: REAL;
	// 轴的纠偏下限
	AxisRecDevPos_L: REAL;
	// 从轴的当前位置
	AxisRecDevActPos: LREAL;
	// 纠偏超限
	PosOverLimit: BOOL;
	// 纠偏传感器上限值
	RecDevSensors_H: REAL;
	// 纠偏传感器下限值
	RecDevSensors_L: REAL;
	// 纠偏轴的速度
	MC_RecDevvelocity: REAL;
	// 纠偏轴的中间速度
	MC_RecDevvelocity_M: REAL;
	// 轴纠偏允许
	MC_RecDevagree: BOOL;
	RecDev_GearInDyn: MC_GearInDyn;
	// 主轴解除耦合

	// 主轴停止
	Master_Stop: MC_Stop;
	// 从轴解除耦合
	SlaveCamOut: MC_CamOut;
	// 主轴匀速运动
	MasterMoveVelocity: MC_MoveVelocity;
	sR_TRIG: R_TRIG;
	sF_TRIG: F_TRIG;
	Slave_Halt: MC_Halt;
	Step0: INT;
	Step3: INT;//双感应器纠偏流程；
	// 主、从轴停止
	AxisStop: BOOL;
	GearInMultiMaster: MC_GearInMultiMaster;
	TON2: TON;
	fRecVlue:REAL;//纠偏值
	fRecAuxVlue:ARRAY [1..10] OF REAL;//纠偏值_辅助
	Error:ARRAY[0..3] OF BOOL;//报警
	bAxisError:BOOL;//
	bFunBlokError:BOOL;//
	
	Riao_K: LREAL;
	step1: INT;
	farrayVlue: ARRAY[0..31] OF REAL;
	i: INT;
	i1: INT;
	i2: INT;
	temp0: REAL;
	cCriterion1: REAL;	// 采集固定的基准值（传感器1）
	cCriterion2: REAL;	// 采集固定的基准值（传感器2）
	// 纠偏传感器1差值；
	sSub1: REAL;
	// 纠偏传感器2差值；
	sSub2: REAL;
	// 双传感器基准偏差值；
	JZData2: REAL;
END_VAR

TON1(IN:= , PT:=T#2S , Q=> , ET=> );//执行延时2S
TON2(IN:=Enable , PT:=T#10S , Q=> , ET=> );//纠偏凸轮耦合超时
sR_TRIG(CLK:=Enable , Q=> );
sF_TRIG(CLK:=Enable , Q=> );

(**************************纠偏传感器的纠偏范围,大于最大值，小于最小值开始纠偏 *****************************)
RecDevSensors_H:=RecDevEqupos1+RecDevValueSet;//纠偏传感器上限值(如果，纠偏传感器的当前值在上、下限这里，就不纠)
RecDevSensors_L:=RecDevEqupos1-RecDevValueSet;//纠偏传感器下限值

(***************************判断纠偏从轴是否超限********************************)	
AxisRecDevPos_H:=AxisintiPos+AxisPos_H;//轴纠偏上限
AxisRecDevPos_L:=AxisintiPos-AxisPos_L;//轴纠偏下限
AxisRecDevActPos:=REAL_TO_LREAL(arrAxisCtrl[SlaveNo].Status.fActPos);

IF bMode=1   THEN
	IF RecDevEqupos1>0 THEN
		IF ABS(RecDevPV1-RecDevEqupos1)>0.2 THEN
			IF RecDevPV1-RecDevEqupos1>0 THEN
				fRecAuxVlue[2]:=0.2;
			ELSE
				fRecAuxVlue[2]:=-0.2;
			END_IF
		ELSE
			fRecAuxVlue[2]:=RecDevPV1-RecDevEqupos1;		
		END_IF
	ELSE
		fRecAuxVlue[2]:=0;
	END_IF
	IF ABS(fRecAuxVlue[2])>recDevValueSet THEN
		fRecVlue:=	fRecAuxVlue[2];
	ELSE
		fRecVlue:=	0;
	END_IF
(*	
//////////////////////////////////////////	
ELSIF bMode=2 THEN
	IF RecDevEqupos1>0 AND RecDevEqupos2>0 THEN
		fRecAuxVlue[1]:=((RecDevPV1-RecDevEqupos1)+(RecDevPV2-RecDevEqupos2))/2 ;
	ELSE
		fRecAuxVlue[1]:=0;
	END_IF
	IF ABS(fRecAuxVlue[1])>recDevValueSet THEN
		fRecVlue:=	fRecAuxVlue[1];
	ELSE
		fRecVlue:=	0;
	END_IF*)
END_IF

IF sStar.Q  THEN
	IF bMode=2 AND cCriterion1>0 AND cCriterion2>0 AND cCriterion1<=9 AND cCriterion2<=9 THEN
			cCriterion1:=RecDevPV1;//固定感应器基准；
			cCriterion2:=RecDevPV2;
	ELSIF bMode=2  AND cCriterion1<=0 OR cCriterion2<=0 OR cCriterion2>9 OR cCriterion2>9 THEN
			JZError[1]:=TRUE;//纠偏传感器位置错误；
	END_IF
END_IF

CASE Step3 OF
10:
IF ModuloActPos >240 AND ModuloActPos <250 THEN
	Step3:=20;
END_IF

20://计算
JZData2:=((cCriterion1-RecDevPV1)+(cCriterion2-RecDevPV2))/2;
	Step3:=23;
	
23://判断极片是否超过93+-0.5范围，超过则不更新基准;
IF JZData2<=0.5 AND JZData2>=-0.5 THEN
	Step3:=25;
ELSE 
	JZError[2]:=TRUE;//感应器测量出误差超限；
	Step3:=27;
END_IF

25://更新最新基准值；这里还是只使用纠偏传感器1的基准来进行调整；
RecDevEqupos1:=(RecDevEqupos1+JZData2)*0.9;//这个需要乘一个系数转移到R角上；系数可以是1，具体看调试的参数是多少合适；
	Step3:=27;
	
27:
	JZData2:=0;
	Step3:=10;
END_CASE
/////////////////////
////////////////////
///////////////////





bReady:= NOT bAxisError  AND NOT bError AND  Step0=0 AND NOT bFunBlokError 
               AND arrAxis[MasterNo].Status.Moving  AND NOT arrAxis[SlaveNo].Status.Coupled  AND arrAxis[SlaveNo].Status.NotMoving
               AND arrAxis[MasterNo].Status.ControlLoopClosed AND arrAxis[SlaveNo].Status.ControlLoopClosed AND
               arrAxis[MasterNo].Status.ConstantVelocity;
			   
CASE Step0 OF
	0://判断使能信号
		IF Enable AND bReady THEN
			Step0:=10;
			TON2.IN:=FALSE;
		END_IF
		IF sF_TRIG.Q THEN
			Step0:=630;
		END_IF
	10://
		IF NOT TON2.Q THEN
			TON2.IN:=TRUE;
			IF arrAxis[SlaveNo].Status.ControlLoopClosed THEN
				TON2.IN:=FALSE;
				Step0:=20;					
			END_IF
		ELSE
				TON2.IN:=FALSE;
				Error[0]:=TRUE;//纠偏凸轮耦合失败
				Step0:=630;	//解耦	
		END_IF
	20://判断从轴是是否耦合，没耦合则启动耦合
			IF GearInMultiMaster.InGear THEN
				Step0:=600;
				bRecOK:=TRUE;
				TON1.IN:=FALSE;	
			ELSE
				GearInMultiMaster.Enable:=TRUE;
			END_IF
	600://从轴纠偏速度计算
			TON1.IN:=TRUE;		
			//IF  TON1.Q THEN //纠偏传感器的当前值 大于 纠偏上限 
				IF NOT PosOverLimit AND  NOT arrAxisCtrl[SlaveNo].Io.biNegLimit AND  NOT arrAxisCtrl[SlaveNo].Io.biPosLimit THEN//判断纠偏是否超限
					MC_RecDevvelocity_M:=fRecVlue*RecDevSpeedCoe;
					IF NOT CWW THEN
						MC_RecDevvelocity:=ScaleTrans(EN:=TRUE , Scalln:=MC_RecDevvelocity_M , X0:=0 , Y0:=0 , X1:=400 , Y1:=10 , Sclofs:=0 );//ScaleTrans的作用是将X0至X1范围之间的输入值，转换为Y0至Y1范围之间的输出值
					ELSE
						MC_RecDevvelocity:=-ScaleTrans(EN:=TRUE , Scalln:=MC_RecDevvelocity_M , X0:=0 , Y0:=0 , X1:=400 , Y1:=10 , Sclofs:=0 );
					END_IF
				ELSIF arrAxisCtrl[SlaveNo].Io.biNegLimit THEN
					Error[1]:=TRUE;//纠偏负限位报警
				ELSIF arrAxisCtrl[SlaveNo].Io.biPosLimit THEN	
					Error[2]:=TRUE;//纠偏正限位报警
				ELSIF PosOverLimit THEN
					Error[3]:=TRUE;//纠偏电机超出设置的纠偏范围	
				END_IF
				IF (Error[1] OR Error[2] OR Error[3] OR bAxisError OR bFunBlokError) OR NOT Enable THEN
					MC_RecDevvelocity:=0;
					Step0:=630;	//解耦	
				END_IF
			//END_IF	
	(******************************  解耦*************************************)
	630:
		 GearInMultiMaster.Enable:=FALSE;    //解除耦合
		 Step0:=640;	
	640:
		 IF   NOT  GearInMultiMaster.InGear  THEN
			 Step0:=650;	
		 END_IF
	650:
		IF arrAxisCtrl[SlaveNo].Status.Coupled THEN
			SlaveCamOut.Execute:=TRUE;
			Step0:=700;
		ELSE
			Step0:=700;	
		END_IF
	700:
		IF NOT arrAxisCtrl[SlaveNo].Status.Coupled   THEN
			SlaveCamOut.Execute:=FALSE;
			bRecOK:=FALSE;
			Slave_Halt.Execute:=TRUE;   
			Step0:=750;	
		END_IF
	750:
		IF arrAxis[SlaveNo].Status.NotMoving  THEN  
			Slave_Halt.Execute:=FALSE;   
		   Step0:=0;  
		END_IF		
END_CASE
	
	
IF RestHMI THEN
	Error[0]:=FALSE;//纠偏凸轮耦合失败
	Error[1]:=FALSE;//纠偏电机负限位报警
	Error[2]:=FALSE;//纠偏电机正限位报警
	Error[3]:=FALSE;//纠偏电机超出设置的纠偏范围
END_IF

bAxisError:=arrAxis[MasterNo].Status.Error OR  arrAxis[SlaveNo].Status.Error ;
bFunBlokError:=GearInMultiMaster.Error OR SlaveCamOut.Error OR Slave_Halt.Error  ;

IF Error[0] OR Error[1] OR Error[2] OR Error[3] OR bAxisError OR bFunBlokError THEN
	bError:=TRUE;
ELSE
	bError:=FALSE;	
END_IF
//纠偏齿轮耦合
IF iMainVel<=60 THEN
	Riao_K:=2;
ELSIF iMainVel>60 AND iMainVel<100 THEN
	Riao_K:=5;
ELSIF iMainVel>=100 AND iMainVel<=120  THEN
	Riao_K:=10;
ELSIF iMainVel>=120 AND iMainVel<=180  THEN
	Riao_K:=15;	
END_IF
IF MasterValue<>0 THEN
	GearInMultiMaster.GearRatio1:=MC_RecDevvelocity/MasterValue*Riao_K;
ELSE
	GearInMultiMaster.GearRatio1:=0;
END_IF
//多主轴耦合，不管主轴的停止还是运行中，都可以耦合从轴
GearInMultiMaster(
	Master1:=arrAxis[MasterNo] , 
	Master2:=arrAxis[SlaveNo] , 
	Master3:=arrAxis[SlaveNo] , 
	Master4:=arrAxis[SlaveNo] , 
	Slave:=arrAxis[SlaveNo]  , 
	Enable:= , 
	GearRatio1:= , 
	GearRatio2:=0 , 
	GearRatio3:=0 , 
	GearRatio4:=0 , 
	Acceleration:= , 
	Deceleration:= , 
	Jerk:= , 
	BufferMode:= , 
	Options:= , 
	InGear=> , 
	Busy=> , 
	Active=> , 
	CommandAborted=> , 
	Error=> , 
	ErrorID=> );
//纠偏从轴解耦
SlaveCamOut(
	Slave:=arrAxis[SlaveNo] , 
	Execute:=, 
	Options:= , 
	Done=> , 
	Busy=> , 
	Error=> , 
	ErrorID=> );
//从轴停止
Slave_Halt(
	Axis:=arrAxis[SlaveNo] , 
	Execute:= , 
	Deceleration:= , 
	Jerk:= , 
	BufferMode:= , 
	Options:= , 
	Done=> , 
	Busy=> , 
	Active=> , 
	CommandAborted=> , 
	Error=> , 
	ErrorID=> );

END_FUNCTION_BLOCK

// ---- POUs/BasicFunction/Data/ScaleTrans.TcPOU
FUNCTION ScaleTrans : REAL
VAR_INPUT
	EN:BOOL;//启动条件
	Scalln:REAL;//输入值
	X0:REAL;//输入范围下限值
	Y0:REAL;//输出范围下限值
	X1:REAL;//输入范围上限值
	Y1:REAL;//输出范围上限值
	Sclofs:REAL;//偏置值
END_VAR
VAR
END_VAR

IF EN THEN
	IF (X1-X0)<> 0 THEN
		ScaleTrans:=(Y1-Y0)/(X1-X0)*(Scalln-X0)+Y0+Sclofs;
	END_IF
END_IF

END_FUNCTION

// ---- POUs/BasicFunction/Basic/07_Ten/FB_TensionVirDriver.TcPOU
FUNCTION_BLOCK FB_TensionVirDriver  //放卷虚轴张力联动
VAR_INPUT
	bReset			       :BOOL;	   
    PidSwitch              :BOOL;	
	fActBufferPos        :REAL;

	fBufferrMinPos	    :REAL;	
	fBufferMaxPos	    :REAL;	
	fBufferBlancePos	:REAL;	
	//fVirMainSpeed       :REAL;
	fWith                   :REAL;
END_VAR

VAR_OUTPUT
	bReady              :BOOL;  
	bTensionOK		 	:BOOL;	
	bError				:BOOL;	
          
END_VAR
VAR_IN_OUT
	virMain		       :axis_ref;		
	TimerAxis	       :axis_ref;	
    Slave		           :axis_ref;		
	bTenExecute		:BOOL;	
END_VAR


VAR


	bAxisError:BOOL;
	rtEnable		:R_TRIG;  
	ftEnable		:F_TRIG;

	TON02: TON;

	rTRIG100: R_TRIG;
	iTensionStep:UINT;


	fbGearOut						:MC_GearOut;		//Unwind
	//fbMoveTimer: MC_MoveVelocity;
	fRatio1: LREAL;
	fRatio2: LREAL;

	fKp2: LREAL;(*乘数系数*)
	Ti: LREAL;
	fbStop: MC_Stop; // Unwind
	bPosLimitError			:BOOL;		
	bNegLimitError			:BOOL;		

	fCalcDancerPos1: REAL;
	fCalcDancerPos2: REAL;

	Delay1,Delay2: TON;
	//bMoveTimer: BOOL;
//	fbhaltTimer: MC_Halt;//TimerAxis


	bFunBlokError: BOOL;

	fMasterLinerSpeed: REAL;
	TM: REAL;
	TM_old: REAL;
	fbGearDync :MC_GearInMultiMaster;
	
	iFlgStart: INT;
	
	bsaveArea: BOOL;
	fTRMax:Tc2_Standard.R_TRIG;
	fTRMin:Tc2_Standard.R_TRIG;
	fTRReset:Tc2_Standard.R_TRIG;	
	bFlgMoveTime:BOOL;
END_VAR

TON02(IN:= , PT:=T#10MS , Q=> , ET=> );

fCalcDancerPos1:=fBufferrMinPos+10;	
fCalcDancerPos2:=fBufferMaxPos-10;

rtEnable(CLK:=bTenExecute , Q=> );        
ftEnable(CLK:=bTenExecute , Q=> );    

bReady:= NOT bAxisError AND NOT bError 
         AND virMain.Status.NotMoving AND TimerAxis.Status.NotMoving AND NOT Slave.Status.Coupled AND Slave.Status.NotMoving
         AND virMain.Status.ControlLoopClosed AND TimerAxis.Status.ControlLoopClosed   AND Slave.Status.ControlLoopClosed ;
		   
IF rtEnable.Q AND bReady THEN
	  iFlgStart:=1;
	  iTensionStep:=100;
ELSIF rtEnable.Q AND NOT bReady THEN	 
   	  bTenExecute:=FALSE;			
ELSIF  ftEnable.Q THEN
     iFlgStart:=2;
     iTensionStep:=100;
END_IF

CASE iTensionStep OF
0:
	fbGearOut.Execute:=FALSE;
	fbStop.Execute:=FALSE;
	bTensionOK:=FALSE;
	TON02.IN:=FALSE;
     iTensionStep:=1;  
1:
  IF bTenExecute AND bReady THEN
    	iTensionStep:=120;  
  END_IF
  IF ftEnable.Q THEN
    	iTensionStep:=630; 
  END_IF


120:  
	 fbGearDync.Enable:=TRUE;    //开启耦合
	 iTensionStep:=550;  
550:
	IF  Slave.Status.Coupled  THEN
		IF   (fActBufferPos<fCalcDancerPos2 AND fActBufferPos>fCalcDancerPos1)    AND PidSwitch    THEN
			bTensionOK:=TRUE;
			iTensionStep:=600;
           ELSIF NOT PidSwitch THEN
			bTensionOK:=TRUE;
			iTensionStep:=600;
		END_IF
	ELSIF fbGearDync.Error OR fbGearDync.CommandAborted   THEN
		  iTensionStep:=630;
	END_IF
(******************************  进入平衡运行阶段   *************************************)
600:
	IF bPosLimitError OR bNegLimitError OR (NOT bTenExecute)  OR bAxisError OR TimerAxis.Status.NotMoving OR NOT Slave.Status.Coupled THEN  
	  TON02.IN:=TRUE;
    ELSIF  ( NOT bTenExecute  OR bAxisError  OR  NOT Slave.Status.Coupled ) AND  NOT  PidSwitch     THEN 
       TON02.IN:=TRUE;
	END_IF
	
	IF TON02.Q THEN   
		IF bPosLimitError  OR  bNegLimitError  OR  bAxisError    THEN
		   bError:=TRUE; 
		END_IF
	    iTensionStep:=630;
	    TON02.IN:=FALSE; 	
	END_IF
	

(******************************  解耦*************************************)
630:
     fbGearDync.Enable:=FALSE;    //开启耦合
     iTensionStep:=635;	
635:
	IF Slave.Status.Coupled THEN
		fbGearOut.Execute:=TRUE;
		iTensionStep:=700;
	ELSE
		iTensionStep:=700;	
	END_IF
700:
	IF NOT Slave.Status.Coupled THEN
		bTensionOK:=FALSE;
		fbStop.Execute:=TRUE;   
		iTensionStep:=750;	
	END_IF
750:
	IF Slave.Status.NotMoving    THEN  
	   fbStop.Execute:=FALSE;
	   iTensionStep:=0;  
	END_IF			
END_CASE



(*********************************** 耦合  *********************************************)
fTRMax(CLK:= fActBufferPos>=  (fBufferBlancePos+fWith/2)   AND bTensionOK , Q=> );  //正极限调节
fTRMin(CLK:= fActBufferPos<=   (fBufferBlancePos-fWith/2)     AND bTensionOK, Q=> );  //负限调节
fTRReset(CLK:= fActBufferPos>=fBufferBlancePos-20 AND fActBufferPos<=fBufferBlancePos+20, Q=> ); //
IF fTRMax.Q OR fTRMin.Q THEN
	bFlgMoveTime:=TRUE;
END_IF
IF fTRReset.Q THEN
	bFlgMoveTime:=FALSE;
END_IF


TM:=2;
fRatio1:=1;//*0.99230769
//fKp2:=SEL(bFlgMoveTime,0,(( fActBufferPos-fBufferBlancePos )*720 ) / (pi*fDriveDiameter*100*TM));//bFlgMoveTime
fKp2:=SEL(bFlgMoveTime,0,(( fActBufferPos-fBufferBlancePos )*720 ) / (fWith*100*TM));
fRatio2:=fKp2;
	

bAxisError:= Slave.Status.Error OR  virMain.Status.Error OR  TimerAxis.Status.Error ;//
bFunBlokError:=fbGearDync.Error OR fbGearOut.Error OR fbStop.Error   ;
rTRIG100(CLK:=bFunBlokError , Q=> );
IF rTRIG100.Q THEN
	bError:=TRUE;
	bTensionOK:=FALSE;
END_IF			
	
IF  bReset AND iTensionStep<>600  AND bError   THEN   //复位处理
    bError:=FALSE;
	iTensionStep:=630;
END_IF

(************************************  张力出错和取消的处理  ******************************************************)
Delay1(IN:=fActBufferPos>fBufferMaxPos AND bTensionOK , PT:=T#300MS , Q=> , ET=> );
bPosLimitError:=Delay1.Q;
Delay2(IN:=fActBufferPos<fBufferrMinPos AND bTensionOK , PT:=T#300MS , Q=> , ET=> );
bNegLimitError:=Delay2.Q;

Motion();

ACTION Motion:
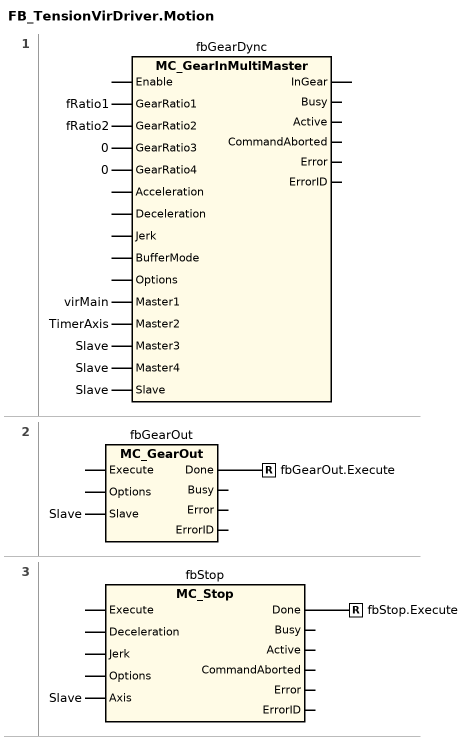
// NETWORK 1
fbGearDync(
    GearRatio1 := fRatio1,
    GearRatio2 := fRatio2,
    GearRatio3 := 0,
    GearRatio4 := 0,
    Master1 := virMain,
    Master2 := TimerAxis,
    Master3 := Slave,
    Master4 := Slave,
    Slave := Slave); // MC_GearInMultiMaster

// NETWORK 2
fbGearOut(Slave := Slave); // MC_GearOut
fbGearOut.Execute R= fbGearOut.Done;

// NETWORK 3
fbStop(Axis := Slave); // MC_Stop
fbStop.Execute R= fbStop.Done;
END_ACTION

END_FUNCTION_BLOCK

// ---- POUs/BasicFunction/User1/FB_CCD_Rounde.TcPOU
FUNCTION_BLOCK FB_CCD_Rounde
VAR_INPUT
	//JzData:REAL;//HMI输入传感器基准值；
	KK:BOOL;//启动开关；
	CCD_Enable: BOOL;//CCD记录启动
	CWW: BOOL;	// 补偿方向选择
	IntervalNum:UINT:=7;//检测机构到执行机构间隔数
	KI_Riao: REAL;		// 补偿系数
	Databace_R3: REAL:=5.5;//R3角工艺杆基准值
	Databace_R4: REAL:=5.5;//R3角工艺杆基准值
	CCD_RoundedSize_R3: REAL;//R3角测量值
	CCD_RoundedSize_R4: REAL;//R4角测量值
	Limt_Max:REAL:=0.1;//补偿上限
	Limt_Min:REAL:=-0.1;//补偿下限
END_VAR
VAR_OUTPUT
		ResultData: REAL;//CCD计算返回结果
END_VAR
VAR_IN_OUT
	JzData:REAL;//HMI输入传感器基准值；
END_VAR


VAR
	STEP0: INT;	
	arrRoundedSize_R3: ARRAY[0..10] OF REAL;//R3数据记录数组
	arrRoundedSize_R4: ARRAY[0..10] OF REAL;//R4数据记录数组
	rCCD_Data: R_TRIG;
	Temp: UINT;
	SumData: REAL;//平均基准值；
	ResultData_1: REAL;
	K1:INT;
	K4:REAL;
	kKs: REAL;// 基准偏差值
	JzData2:REAL;
END_VAR

VAR CONSTANT
	//Num: UINT:=10;//采集次数
END_VAR

IF KK THEN //开关；

rCCD_Data(CLK:=CCD_Enable , Q=> );//CCD记录数据开始
CASE STEP0 OF
	
0://启动CCD拍照，记录R角纵深的数据
			MEMSET(ADR(arrRoundedSize_R3),0,SIZEOF(arrRoundedSize_R3)); 
			MEMSET(ADR(arrRoundedSize_R4),0,SIZEOF(arrRoundedSize_R4)); 
			JzData2:=0;
			kKs:=0;			
			SumData:=0;
			Temp:=0;                                                                                                                                                                                                                                                                                                                                                                                             
			K4:=0;
			FOR K1:=1 TO 10BY 1 DO 	
				arrRoundedSize_R3[K1]:=0;
				arrRoundedSize_R4[K1]:=0;
			END_FOR
			STEP0:=10;
10://尺寸检测OK,开始记录CCD  R角数据
				IF rCCD_Data.Q AND  CCD_RoundedSize_R4>=Databace_R4-1.2 AND  CCD_RoundedSize_R4<Databace_R4+1.2 THEN//+-1.2 采集的数据范围，这里可以比红线再外一些，可以包括NG数据，但是那种很明显尺寸太大或者太小的数据就不要；
					Temp:=Temp+1;
					IF Temp<=10  THEN//采集10个数据；
						arrRoundedSize_R3[Temp]:=CCD_RoundedSize_R3;//非极耳则的R角数据
						arrRoundedSize_R4[Temp]:=CCD_RoundedSize_R4;//极耳则的R角数据
					ELSE
						STEP0:=20;
					END_IF
				END_IF				
						
20://求平均值；
			SumData:=(arrRoundedSize_R4[1]+arrRoundedSize_R4[2]+arrRoundedSize_R4[3]+arrRoundedSize_R4[4]+arrRoundedSize_R4[5]+arrRoundedSize_R4[6]+arrRoundedSize_R4[7]+arrRoundedSize_R4[8]+arrRoundedSize_R4[9])/9;
				IF SumData>=1 THEN//不为零；																															
					STEP0:=30;					
				END_IF

30://判断是否需要校准曲线；
kKs:=SumData-Databace_R4;//kKs:=SumData-5.5;
	IF kKs<=0.08 AND  kKs>=-0.08  THEN//曲线与基准值重合；不校准；
		STEP0:=0;
	END_IF
	
	IF kKs>0.08 OR kKs<-0.08  THEN//曲线需要校准；
		STEP0:=33;
	END_IF

33://纠偏系数分级；
IF kKs>=0.8 OR kKs<=-0.8 THEN
	K4:=JzData-(kKs*0.8);
END_IF

IF kKs>=0.4 AND kKs<0.8 OR kKs<=-0.4 AND kKs>-0.8 THEN
	K4:=JzData-(kKs*0.6);
END_IF

IF  kKs<0.4 AND kKs>-0.4 THEN
	K4:=JzData-(kKs*0.4);
END_IF
	STEP0:=37;	
	
37:
IF K4<=Databace_R4+1.0 AND K4>=Databace_R4-1.0 THEN//计算出的基准值不在范围内则该周期不进行调整基准值；或者给一个固定值5.3和2.2；
	JzData2:=K4;
	STEP0:=39;	
ELSE
//	STEP0:=50;//给固定值；
	STEP0:=0;//不校准或者报警；
END_IF
(*
50:
	IF K4>Databace_R3 THEN
		JzData2:=4.0;
	END_IF

	IF K4<2.0  THEN
		JzData2:=3.0 ;
	END_IF
STEP0:=39;
	*)
39://输入最新的基准值；
IF JzData2<>0 THEN
		JzData:=JzData2;
		STEP0:=0;	
END_IF	

END_CASE
END_IF

END_FUNCTION_BLOCK

// ---- POUs/BasicFunction/Data/FB_ProductionDataLocal.TcPOU
FUNCTION_BLOCK FB_ProductionDataLocal

VAR_INPUT
	NowTimeData	:TIMESTRUCT;(*当前系统时间*)
	OutFlag1:BOOL;(*产量计数标志1*)
	OutFlag2:BOOL;(*产量计数标志2*)
	NGFlag:ARRAY[1..50] OF BOOL;(*NG计数标志*)

	RunFlag:BOOL;(*运行标志*)
	WaitFlag:BOOL;(*待料标志*)
	AlarmFlag:BOOL;(*故障标志*)
	DelDataAMBtn:BOOL;(*白班数据清除按钮*)
	DelDataPMBtn:BOOL;(*夜班数据清除按钮*)
	NGClearAMBtn:ARRAY[1..50] OF BOOL;//白班NG类型计数清零
	NGClearPMBtn:ARRAY[1..50] OF BOOL;//夜班NG类型计数清零
END_VAR



VAR_OUTPUT
	NowOutTotal:REAL;(*当前班次加工总数*)
	NowRate:REAL;(*当前班次良率*)
	OEE:REAL;//稼动率
END_VAR

VAR_IN_OUT
	NowDay				:INT;(*数据移位时所保存当前日*)
	NowMonth			:INT;(*数据移位时所保存当前月*)
	DayHistory			:ARRAY[1..7 ] 	OF INT;(*历史日*)
	MonthHistory		:ARRAY[1..7 ] 	OF INT;(*历史月*)
	TodayTotal:REAL;(*当天24H生产总数*)
	TodayOK:REAL;(*当天24H生产OK总数*)
	TodayNG:REAL;(*当天24H生产NG总数*)
	TodayTotal_AM:REAL;(*当天白班生产总数*)
	TodayTotal_PM:REAL;(*当天夜班生产总数*)
	TodayRate_AM:REAL;(*当天白班良率*)
	TodayRate_PM:REAL;(*当天夜班良率*)
	TodayOK_AM:REAL;(*当天白班生产OK总数*)
	TodayOK_PM:REAL;(*当天夜班生产OK总数*)
	TodayNG_AM:REAL;(*当天白班生产NG总数*)
	TodayNG_PM:REAL;(*当天夜班生产NG总数*)
	TodayHour_AM		:ARRAY[8..19 ] 	OF REAL;(*当天白班每小时产量ARRAY[8..19 ]*)
	TodayHour_PM		:ARRAY[0..23] 	OF REAL;(*当天夜班每小时产量ARRAY[0..23]*)
	TodayNGClass_AM		:ARRAY[1..50 ] 	OF REAL;(*当天白班各类NG数量ARRAY[1..30 ]*)
	TodayNGClass_PM		:ARRAY[1..50 ] 	OF REAL;(*当天夜班各类NG数量ARRAY[1..30 ]*)
	TodayRun_AM			:REAL;(*当天白班总运行时间合计/分*)
	TodayRun_PM			:REAL;(*当天夜班总运行时间合计/分*)
	TodayWait_AM		:REAL;(*当天白班总待料时间合计/分*)
	TodayWait_PM		:REAL;(*当天夜班总待料时间合计/分*)
	TodayAlarm_AM		:REAL;(*当天白班总报警时间合计/分*)
	TodayAlarm_PM		:REAL;(*当天夜班总报警时间合计/分*)

	RunCnt_AM:ARRAY[8..19 ] 	OF UDINT;	(*白班运行时间计数*)
	RunCnt_PM:ARRAY[0..23] 		OF UDINT;	(*夜班运行时间计数*)
	WaitCnt_AM:ARRAY[8..19 ] 	OF UDINT;	(*白班待料时间计数*)
	WaitCnt_PM:ARRAY[0..23] 	OF UDINT;	(*夜班待料时间计数*)
	AlarmCnt_AM:ARRAY[8..19 ] 	OF UDINT;	(*白班报警时间计数*)
	AlarmCnt_PM:ARRAY[0..23] 	OF UDINT;	(*夜班报警时间计数*)

	TodayRun_AMH:ARRAY[8..19 ] OF REAL;(*当天白班每小时运行时间合计/分*)
	TodayRun_PMH:ARRAY[0..23]OF REAL;(*当天夜班每小时运行时间合计/分*)
	TodayWait_AMH:ARRAY[8..19 ] OF REAL;(*当天白班每小时待料时间合计/分*)
	TodayWait_PMH:ARRAY[0..23]OF REAL;(*当天夜班每小时待料时间合计/分*)
	TodayAlarm_AMH	:ARRAY[8..19 ] 	OF	REAL;(*当天白班每小时报警时间合计/分*)
	TodayAlarm_PMH	:ARRAY[0..23]OF REAL;(*当天夜班每小时报警时间合计/分*)

	HistoryTotal:ARRAY[1..7 ] OF REAL;(*历史每天24H生产总数ARRAY[1..7 ]*)
	HistoryOK:ARRAY[1..7 ] OF REAL;(*历史每天24H生产OK总数ARRAY[1..7 ]*)
	HistoryNG:ARRAY[1..7 ] OF REAL;(*历史每天24H生产NG总数ARRAY[1..7 ]*)
	HistoryTotal_AM:ARRAY[1..7 ] OF REAL;(*历史每天白班生产总数ARRAY[1..7 ]*)
	HistoryTotal_PM:ARRAY[1..7 ] OF REAL;(*历史每天夜班生产总数ARRAY[1..7 ]*)
	HistoryRate_AM:ARRAY[1..7 ] OF REAL;(*历史每天白班良率ARRAY[1..7 ]*)
	HistoryRate_PM:ARRAY[1..7 ] OF REAL;(*历史每天夜班良率ARRAY[1..7 ]*)
	HistoryOK_AM:ARRAY[1..7 ] OF REAL;(*历史每天白班生产OK总数ARRAY[1..7 ]*)
	HistoryOK_PM:ARRAY[1..7 ] OF REAL;(*历史每天夜班生产OK总数ARRAY[1..7 ]*)
	HistoryNG_AM:ARRAY[1..7 ] OF REAL;(*历史每天白班生产NG总数ARRAY[1..7 ]*)
	HistoryNG_PM:ARRAY[1..7 ] OF REAL;(*历史每天夜班生产NG总数ARRAY[1..7 ]*)
	HistoryHour_AM		:ARRAY[1..7,8..19 ] 	OF REAL;(*历史每天白班每小时产量ARRAY[1..7,8..19 ]*)
	HistoryHour_PM		:ARRAY[1..7,0..23] 		OF REAL;(*历史每天夜班每小时产量ARRAY[1..7,0..23]*)
	HistoryNGClass_AM	:ARRAY[1..7,1..50 ] 	OF REAL;(*历史每天白班各类NG数量ARRAY[1..7,1..30 ]*)
	HistoryNGClass_PM	:ARRAY[1..7,1..50 ] 	OF REAL;(*历史每天夜班各类NG数量ARRAY[1..7,1..30 ]*)
	HistoryRun_AM		:ARRAY[1..7 ] OF REAL;(*历史每天白班总运行时间合计ARRAY[1..7 ]*)
	HistoryRun_PM		:ARRAY[1..7 ] OF REAL;(*历史每天夜班总运行时间合计ARRAY[1..7 ]*)
	HistoryWait_AM		:ARRAY[1..7 ] OF REAL;(*历史每天白班总待料时间合计ARRAY[1..7 ]*)
	HistoryWait_PM		:ARRAY[1..7 ] OF REAL;(*历史每天夜班总待料时间合计ARRAY[1..7 ]*)
	HistoryAlarm_AM		:ARRAY[1..7 ] OF REAL;(*历史每天白班总报警时间合计ARRAY[1..7 ]*)
	HistoryAlarm_PM		:ARRAY[1..7 ] OF REAL;(*历史每天夜班总报警时间合计ARRAY[1..7 ]*)

	HistoryRun_AMH		:ARRAY[1..7,8..19 ] OF REAL;(*历史每天白班每小时运行时间合计ARRAY[1..7 ]*)
	HistoryRun_PMH		:ARRAY[1..7,0..23 ] OF REAL;(*历史每天夜班每小时运行时间合计ARRAY[1..7 ]*)
	HistoryWait_AMH		:ARRAY[1..7,8..19 ] OF REAL;(*历史每天白班每小时待料时间合计ARRAY[1..7 ]*)
	HistoryWait_PMH		:ARRAY[1..7,0..23 ] OF REAL;(*历史每天夜班每小时待料时间合计ARRAY[1..7 ]*)
	HistoryAlarm_AMH	:ARRAY[1..7,8..19 ] OF REAL;(*历史每天白班每小时报警时间合计ARRAY[1..7 ]*)
	HistoryAlarm_PMH	:ARRAY[1..7,0..23 ] OF REAL;(*历史每天夜班每小时报警时间合计ARRAY[1..7 ]*)
	
	TodayNgHour_Day:ARRAY[1..50,0..23] OF REAL;//白班每小时NG类型统计,,
	TodayNgHour_Night:ARRAY[1..50,0..23] OF REAL;//夜班每小时NG类型统计,,
	HisTodayNgHour_Day:ARRAY[1..50,0..23,1..7] OF REAL;//l历史白班每小时NG类型统计,,
	HisTodayNgHour_Night:ARRAY[1..50,0..23,1..7] OF REAL;//历史夜班每小时NG类型统计,,			
		
	TodayNGQualified:ARRAY[1..50] OF REAL;//当天白班各种NG类型NG率
	NightNGQualified:ARRAY[1..50] OF REAL;//当天夜班各种NG类型NG率	
	
	HisTodayNGQualified:ARRAY[1..50,1..7] OF REAL;//历史白班各种NG类型NG率
	HisNightNGQualified:ARRAY[1..50,1..7] OF REAL;//历史夜班各种NG类型NG率
END_VAR


VAR
	i:INT;
	j: INT;
	K:INT;
	m:INT;
	d:INT;
	TrigOutAdd1:R_TRIG ;	(*产量计数上升沿1*)
	TrigOutAdd2:R_TRIG ;	(*产量计数上升沿1*)
	TrigNgAdd: ARRAY[1..50 ] OF R_TRIG;(*1-30类ng计数统计*)
	HistoryData_Step:UINT;(*历史数据保存步*)
	SaveDataDelay:TON;(*历史数据保存延时，防止处理周期内多次存储*)
	rNGClearAMBtn:ARRAY [1..50] OF R_TRIG;//白班ng类型清零上升沿
	rNGClearPMBtn:ARRAY [1..50] OF R_TRIG;//夜班NG类型清零上升沿
END_VAR


(**********************  分段产能  ***************************************)
TrigOutAdd1(CLK:=OutFlag1,Q=> );(*产量计数上升沿1*)
TrigOutAdd2(CLK:=OutFlag2,Q=> );(*产量计数上升沿1*)
FOR i:=1 TO 50 DO
	rNGClearAMBtn[i](CLK:=NGClearAMBtn[i],Q=> );//白班ng类型清零上升沿
	rNGClearPMBtn[i](CLK:=NGClearPMBtn[i],Q=> );//夜班NG类型清零上升沿
END_FOR
FOR m:=1 TO 50 DO
	IF  rNGClearAMBtn[m].Q THEN
		TodayNGClass_AM[m]:=0;
		TodayNGQualified[m]:=0;
	END_IF
	IF  rNGClearPMBtn[m].Q THEN
		TodayNGClass_PM[m]:=0;
		NightNGQualified[m]:=0;
	END_IF
END_FOR

//NG分类统计触发
TrigNgAdd[1](CLK:=NGFlag[1],Q=> );(*1类ng*)//极片长度不良
TrigNgAdd[2](CLK:=NGFlag[2],Q=> );(*2类ng*)//极片CIL宽度不良
TrigNgAdd[3](CLK:=NGFlag[3],Q=> );(*3类ng*)//极片宽度不良
TrigNgAdd[4](CLK:=NGFlag[4],Q=> );(*4类ng*)//极耳宽度不良
TrigNgAdd[5](CLK:=NGFlag[5],Q=> );(*5类ng*)//极耳高度不良
TrigNgAdd[6](CLK:=NGFlag[6],Q=> );(*6类ng*)//极耳侧边距不良
TrigNgAdd[7](CLK:=NGFlag[7],Q=> );(*7类ng*)//极耳面积不良
TrigNgAdd[8](CLK:=NGFlag[8],Q=> );(*8类ng*)//圆角深度不良
TrigNgAdd[9](CLK:=NGFlag[9],Q=> );(*9类ng*)//极耳边缘角度不良
TrigNgAdd[10](CLK:=NGFlag[10],Q=> );(*10类ng*)//圆角宽度不良
TrigNgAdd[11](CLK:=NGFlag[11],Q=> );(*11类ng*)//圆角轮廓不良
TrigNgAdd[12](CLK:=NGFlag[12],Q=> );(*12类ng*)//圆角面积不良
TrigNgAdd[13](CLK:=NGFlag[13],Q=> );(*13类ng*)//圆角余料不良
TrigNgAdd[14](CLK:=NGFlag[14],Q=> );(*14类ng*)//尺寸其他不良
TrigNgAdd[15](CLK:=NGFlag[15],Q=> );(*15类ng*)//来料极耳间距不良
TrigNgAdd[16](CLK:=NGFlag[16],Q=> );(*16类ng*)
TrigNgAdd[17](CLK:=NGFlag[17],Q=> );(*17类ng*)
TrigNgAdd[18](CLK:=NGFlag[18],Q=> );(*18类ng*)
TrigNgAdd[19](CLK:=NGFlag[19],Q=> );(*19类ng*)
TrigNgAdd[20](CLK:=NGFlag[20],Q=> );(*20类ng*)
TrigNgAdd[21](CLK:=NGFlag[21],Q=> );(*21类ng*)//抓边失败
TrigNgAdd[22](CLK:=NGFlag[22],Q=> );(*22类ng*)//直边不良标志位
TrigNgAdd[23](CLK:=NGFlag[23],Q=> );(*23类ng*)//极片缺失
TrigNgAdd[24](CLK:=NGFlag[24],Q=> );(*24类ng*)//接带
TrigNgAdd[25](CLK:=NGFlag[25],Q=> );(*25类ng*)//线扫黄标
TrigNgAdd[26](CLK:=NGFlag[26],Q=> );(*26类ng*)//漏金属
TrigNgAdd[27](CLK:=NGFlag[27],Q=> );(*27类ng*)//气泡
TrigNgAdd[28](CLK:=NGFlag[28],Q=> );(*28类ng*)//暗条痕
TrigNgAdd[29](CLK:=NGFlag[29],Q=> );(*29类ng*)//亮条痕
TrigNgAdd[30](CLK:=NGFlag[30],Q=> );(*30类ng*)//破损
TrigNgAdd[31](CLK:=NGFlag[31],Q=> );(*31类ng*)//碎屑
TrigNgAdd[32](CLK:=NGFlag[32],Q=> );(*32类ng*)//通讯超时
TrigNgAdd[33](CLK:=NGFlag[33],Q=> );(*33类ng*)//脱碳
TrigNgAdd[34](CLK:=NGFlag[34],Q=> );(*34类ng*)//其他
TrigNgAdd[35](CLK:=NGFlag[35],Q=> );(*35类ng*)
TrigNgAdd[36](CLK:=NGFlag[36],Q=> );(*36类ng*)
TrigNgAdd[37](CLK:=NGFlag[37],Q=> );(*37类ng*)
TrigNgAdd[38](CLK:=NGFlag[38],Q=> );(*38类ng*)
TrigNgAdd[39](CLK:=NGFlag[39],Q=> );(*39类ng*)
TrigNgAdd[40](CLK:=NGFlag[40],Q=> );(*40类ng*)
TrigNgAdd[41](CLK:=NGFlag[41],Q=> );(*41类ng*)
TrigNgAdd[42](CLK:=NGFlag[42],Q=> );(*42类ng*)
TrigNgAdd[43](CLK:=NGFlag[43],Q=> );(*43类ng*)//接带计数
TrigNgAdd[44](CLK:=NGFlag[44],Q=> );(*44类ng*)//黄标跳切计数
TrigNgAdd[45](CLK:=NGFlag[45],Q=> );(*45类ng*)//黄标计数
TrigNgAdd[46](CLK:=NGFlag[46],Q=> );(*46类ng*)
TrigNgAdd[47](CLK:=NGFlag[47],Q=> );(*47类ng*)
TrigNgAdd[48](CLK:=NGFlag[48],Q=> );(*48类ng*)//线扫NG数
TrigNgAdd[49](CLK:=NGFlag[49],Q=> );(*49类ng*)//尺寸NG数
TrigNgAdd[50](CLK:=NGFlag[50],Q=> );(*50类ng*)//

(***白班数据统计******)
FOR i:=8 TO 19 DO
	IF NowTimeData.wHour=i THEN
		IF i>=8 AND i<=19 THEN
			(********产量计数**********)
			IF TrigOutAdd1.Q  THEN
				TodayHour_AM[i]:=TodayHour_AM[i]+1;
			END_IF
			IF TrigOutAdd2.Q  THEN
				TodayHour_AM[i]:=TodayHour_AM[i]+1;
			END_IF
			(*******白班NG不良分类统计*)
			FOR m:=1 TO 50 DO
				IF TrigNgAdd[m].Q THEN
					TodayNGClass_AM[m]:=TodayNGClass_AM[m]+1;
				END_IF 
				(*
				IF  rNGClearAMBtn[m].Q THEN
					TodayNGClass_AM[m]:=0;
				END_IF
				*)
			END_FOR
			(******************白班每小时NG类型统计*******************)
			FOR m:=1 TO 50 DO
				IF TrigNgAdd[m].Q THEN
					TodayNgHour_Day[m,i]:=TodayNgHour_Day[m,i]+1;//白班每小时NG类型统计
				END_IF
			END_FOR
			
			 (*运行时间统计*)
			IF RunFlag THEN
				RunCnt_AM[i]:=RunCnt_AM[i]+1;
			END_IF
			IF RunCnt_AM[i] <>0 THEN
				TodayRun_AMH[i]:=UDINT_TO_REAL(RunCnt_AM[i]/(500*60)) ;
			END_IF
			
			 (*待料时间统计*)
			IF  WaitFlag  THEN
				WaitCnt_AM[i]:=WaitCnt_AM[i]+1;
			END_IF
			IF WaitCnt_AM[i]<>0 THEN
				TodayWait_AMH[i]:=UDINT_TO_REAL(WaitCnt_AM[i]/(500*60)) ;
			END_IF
			(*报警时间统计*)
			IF  AlarmFlag THEN
				AlarmCnt_AM[i]:=AlarmCnt_AM[i]+1;
			END_IF
			IF AlarmCnt_AM[i]<>0 THEN
				TodayAlarm_AMH[i]:=UDINT_TO_REAL(AlarmCnt_AM[i]/(500*60)) ;
			END_IF
			(*当前生产输出*)
			NowOutTotal:=TodayTotal_AM;
			NowRate:=TodayRate_AM;
			
			
			//欣旺达个性生产数据
			IF TodayTotal_AM<>0 THEN
				FOR k:=1 TO 50 DO
					TodayNGQualified[k]:=100*(TodayNGClass_AM[k]/TodayTotal_AM);//当天夜班尺寸NG率
				END_FOR
			END_IF
		
			
		END_IF
	END_IF
END_FOR

(***手动清除白班产量统计数据******)
IF DelDataAMBtn THEN
	FOR m:=1 TO 50 DO
		TodayNGQualified[m]:=0;
		TodayNGClass_AM[m]:=0;
	END_FOR
	FOR j := 8 TO 19 DO
		TodayHour_AM[j]:=0 ;
		RunCnt_AM[j]:= 0 ;(*白班运行时间计数*)
		AlarmCnt_AM[j]:= 0 ;(*白班报警时间计数*)
		WaitCnt_AM[j]:= 0 ;(*白班待料时间计数*)
		
		RunCnt_AM[j]:=0;
		TodayRun_AMH[j]:=0;
		WaitCnt_AM[j]:=0;
		TodayWait_AMH[j]:=0;
		AlarmCnt_AM[j]:=0;
		TodayAlarm_AMH[j]:=0;
		FOR d:=1 TO 50 DO
			TodayNgHour_Day[d,j]:=0;
			TodayNGQualified[d]:=0;
		END_FOR
	END_FOR
	(*
	FOR j := 1 TO 20 DO
		TodayNGClass_AM[j] := 0 ;
	END_FOR
	*)
	TodayTotal_AM:=0;(*当天白班生产总数*)
	TodayRate_AM:=0;(*当天白班良率*)
	TodayOK_AM:=0;(*当天白班生产OK总数*)
	TodayNG_AM:=0;(*当天白班生产NG总数*)
	
END_IF
(*当天白班生产总数*)
TodayTotal_AM:=TodayHour_AM[8]+TodayHour_AM[9]+TodayHour_AM[10]+TodayHour_AM[11]+TodayHour_AM[12]+TodayHour_AM[13]+
				TodayHour_AM[14]+TodayHour_AM[15]+TodayHour_AM[16]+TodayHour_AM[17]+TodayHour_AM[18]+TodayHour_AM[19];
(*当天白班生产NG总数*)
TodayNG_AM:=TodayNGClass_AM[1]+TodayNGClass_AM[2]+TodayNGClass_AM[3]+TodayNGClass_AM[4]+TodayNGClass_AM[5]+
				TodayNGClass_AM[6]+TodayNGClass_AM[7]+TodayNGClass_AM[8]+TodayNGClass_AM[9]+TodayNGClass_AM[10]+
				TodayNGClass_AM[11]+TodayNGClass_AM[12]+TodayNGClass_AM[13]+TodayNGClass_AM[14]+(*TodayNGClass_AM[15]+*)
				TodayNGClass_AM[16]+TodayNGClass_AM[17]+TodayNGClass_AM[18]+TodayNGClass_AM[19]+TodayNGClass_AM[20]+
				TodayNGClass_AM[21]+TodayNGClass_AM[22]+TodayNGClass_AM[23]+TodayNGClass_AM[24]+TodayNGClass_AM[25]+
				TodayNGClass_AM[26]+TodayNGClass_AM[27]+TodayNGClass_AM[28]+TodayNGClass_AM[29]+TodayNGClass_AM[30]+
				TodayNGClass_AM[31]+TodayNGClass_AM[32]+TodayNGClass_AM[33]+TodayNGClass_AM[34]+TodayNGClass_AM[35];
(*当天白班生产OK总数*)
TodayOK_AM:=TodayTotal_AM-TodayNG_AM;
(*当天白班良率*)
IF TodayTotal_AM<>0 THEN
	TodayRate_AM:=100*TodayOK_AM/TodayTotal_AM;
END_IF

(*当天白班总运行时间合计/分*)
TodayRun_AM:=TodayRun_AMH[8]+TodayRun_AMH[9]+TodayRun_AMH[10]+TodayRun_AMH[11]+TodayRun_AMH[12]+TodayRun_AMH[13]+
				TodayRun_AMH[14]+TodayRun_AMH[15]+TodayRun_AMH[16]+TodayRun_AMH[17]+TodayRun_AMH[18]+TodayRun_AMH[19];
(*当天白班总待料时间合计/分*)
TodayWait_AM:=TodayWait_AMH[8]+TodayWait_AMH[9]+TodayWait_AMH[10]+TodayWait_AMH[11]+TodayWait_AMH[12]+TodayWait_AMH[13]+
				TodayWait_AMH[14]+TodayWait_AMH[15]+TodayWait_AMH[16]+TodayWait_AMH[17]+TodayWait_AMH[18]+TodayWait_AMH[19];
(*当天白班总报警时间合计/分*)
TodayAlarm_AM:=TodayAlarm_AMH[8]+TodayAlarm_AMH[9]+TodayAlarm_AMH[10]+TodayAlarm_AMH[11]+TodayAlarm_AMH[12]+TodayAlarm_AMH[13]+
				TodayAlarm_AMH[14]+TodayAlarm_AMH[15]+TodayAlarm_AMH[16]+TodayAlarm_AMH[17]+TodayAlarm_AMH[18]+TodayAlarm_AMH[19];
(***白班数据统计******)


(*******夜班数据统计******)
FOR i:=0 TO 23 DO
	IF NowTimeData.wHour=i THEN
		IF i<=7 OR i>=20 THEN
			(********产量计数**********)
			IF TrigOutAdd1.Q  THEN
				TodayHour_PM[i]:=TodayHour_PM[i]+1;
			END_IF
			IF TrigOutAdd2.Q  THEN
				TodayHour_PM[i]:=TodayHour_PM[i]+1;
			END_IF
			(*******夜班NG不良分类统计*)
			FOR m:= 1 TO 50 DO
				IF TrigNgAdd[m].Q THEN
					TodayNGClass_PM[m]:=TodayNGClass_PM[m]+1;
				END_IF
				(*
				IF  rNGClearPMBtn[m].Q THEN
					TodayNGClass_PM[m]:=0;
				END_IF
				*)
			END_FOR
			(******************夜班每小时NG类型统计*******************)
			FOR m:= 1 TO 50 DO
				IF TrigNgAdd[m].Q THEN
					TodayNgHour_Night[m,i]:=TodayNgHour_Night[m,i]+1;//夜班每小时NG类型统计
				END_IF
			END_FOR
			 (*运行时间统计*)
			IF RunFlag THEN
				RunCnt_PM[i]:=RunCnt_PM[i]+1;
			END_IF
			IF RunCnt_PM[i]<>0 THEN
				TodayRun_PMH[i]:=UDINT_TO_REAL(RunCnt_PM[i]/(500*60)) ;
			END_IF
			 (*待料时间统计*)
			IF  WaitFlag  THEN
				WaitCnt_PM[i]:=WaitCnt_PM[i]+1;
			END_IF
			IF WaitCnt_PM[i]<>0 THEN
				TodayWait_PMH[i]:=UDINT_TO_REAL(WaitCnt_PM[i]/(500*60)) ;
			END_IF
			(*报警时间统计*)
			IF  AlarmFlag THEN
				AlarmCnt_PM[i]:=AlarmCnt_PM[i]+1;
			END_IF
			IF AlarmCnt_PM[i]<>0 THEN
				TodayAlarm_PMH[i]:=UDINT_TO_REAL(AlarmCnt_PM[i]/(500*60)) ;
			END_IF
			(*当前生产输出*)
			NowOutTotal:=TodayTotal_PM;
			NowRate:=TodayRate_PM;
			
			//欣旺达个性生产数据
			IF TodayTotal_PM<>0 THEN
				FOR k:=1 TO 50 DO
					NightNGQualified[k]:=100*(TodayNGClass_PM[k]/TodayTotal_PM);//当天夜班尺寸NG率
				END_FOR
			END_IF
		END_IF
	END_IF
END_FOR

(***手动清除夜班产量统计数据******)
IF DelDataPMBtn THEN
	FOR m:=1 TO 50 DO
		NightNGQualified[m]:=0;
		TodayNGClass_PM[m]:=0;
	END_FOR
	FOR j:=0 TO 23 DO
		TodayHour_PM[j]:=0 ;
		RunCnt_PM[j]:= 0 ;(*夜班运行时间计数*)
		AlarmCnt_PM[j]:=0;(*夜班报警时间计数*)
		WaitCnt_PM[j]:= 0 ;(*夜班待料时间计数*)
		RunCnt_PM[j]:=0;
		TodayRun_PMH[j]:=0;
		WaitCnt_PM[j]:=0;
		TodayWait_PMH[j]:=0;
		AlarmCnt_PM[j]:=0;
		TodayAlarm_PMH[j]:=0;
		FOR d:=1 TO 50 DO
			TodayNgHour_Night[d,j]:=0;
		END_FOR
(*
	FOR j := 1 TO 20 DO
		TodayNGClass_PM[j] := 0 ;
	END_FOR
*)
	TodayTotal_PM:=0;(*当天夜班生产总数*)
	TodayRate_PM:=0;(*当天夜班良率*)
	TodayOK_PM:=0;(*当天夜班生产OK总数*)
	TodayNG_PM:=0;(*当天夜班生产NG总数*)
	END_FOR
END_IF

(*当天夜班生产总数*)
TodayTotal_PM:=TodayHour_PM[20]+TodayHour_PM[21]+TodayHour_PM[22]+TodayHour_PM[23]+TodayHour_PM[0]+TodayHour_PM[1]+
					TodayHour_PM[2]+TodayHour_PM[3]+TodayHour_PM[4]+TodayHour_PM[5]+TodayHour_PM[6]+TodayHour_PM[7];
(*当天夜班生产NG总数*)
TodayNG_PM:=TodayNGClass_PM[1]+TodayNGClass_PM[2]+TodayNGClass_PM[3]+TodayNGClass_PM[4]+TodayNGClass_PM[5]+
				TodayNGClass_PM[6]+TodayNGClass_PM[7]+TodayNGClass_PM[8]+TodayNGClass_PM[9]+TodayNGClass_PM[10]+
				TodayNGClass_PM[11]+TodayNGClass_PM[12]+TodayNGClass_PM[13]+TodayNGClass_PM[14]+(*TodayNGClass_PM[15]+*)
				TodayNGClass_PM[16]+TodayNGClass_PM[17]+TodayNGClass_PM[18]+TodayNGClass_PM[19]+TodayNGClass_PM[20]+
				TodayNGClass_PM[21]+TodayNGClass_PM[22]+TodayNGClass_PM[23]+TodayNGClass_PM[24]+TodayNGClass_PM[25]+
				TodayNGClass_PM[26]+TodayNGClass_PM[27]+TodayNGClass_PM[28]+TodayNGClass_PM[29]+TodayNGClass_PM[30]+
				TodayNGClass_PM[31]+TodayNGClass_PM[32]+TodayNGClass_PM[33]+TodayNGClass_PM[34]+TodayNGClass_PM[35];
(*当天夜班生产OK总数*)
TodayOK_PM:=TodayTotal_PM-TodayNG_PM;
(*当天夜班良率*)
IF TodayTotal_PM<>0 THEN
	TodayRate_PM:=100*TodayOK_PM/TodayTotal_PM;
END_IF
(*当天夜班总运行时间合计/分*)
TodayRun_PM:=TodayRun_PMH[20]+TodayRun_PMH[21]+TodayRun_PMH[22]+TodayRun_PMH[23]+TodayRun_PMH[0]+TodayRun_PMH[1]+
			TodayRun_PMH[2]+TodayRun_PMH[3]+TodayRun_PMH[4]+TodayRun_PMH[5]+TodayRun_PMH[6]+TodayRun_PMH[7];
(*当天夜班总待料时间合计/分*)
TodayWait_PM:=TodayWait_PMH[20]+TodayWait_PMH[21]+TodayWait_PMH[22]+TodayWait_PMH[23]+TodayWait_PMH[0]+TodayWait_PMH[1]+
			TodayWait_PMH[2]+TodayWait_PMH[3]+TodayWait_PMH[4]+TodayWait_PMH[5]+TodayWait_PMH[6]+TodayWait_PMH[7];
(*当天夜班总报警时间合计/分*)
TodayAlarm_PM:=TodayAlarm_PMH[20]+TodayAlarm_PMH[21]+TodayAlarm_PMH[22]+TodayAlarm_PMH[23]+TodayAlarm_PMH[0]+TodayAlarm_PMH[1]+
			TodayAlarm_PMH[2]+TodayAlarm_PMH[3]+TodayAlarm_PMH[4]+TodayAlarm_PMH[5]+TodayAlarm_PMH[6]+TodayAlarm_PMH[7];

(*******夜班数据统计******)


(*******白班+夜班数据汇总******)
TodayTotal:=TodayTotal_AM+TodayTotal_PM;(*当天生产总数*)
TodayNG:=TodayNG_AM+TodayNG_PM;(*当天生产NG总数*)
TodayOK:=TodayTotal-TodayNG;(*当天生产OK总数*)
(*******白班+夜班数据汇总******)


(*************历史数据存储**************)
CASE HistoryData_Step OF
0:
	IF NowTimeData.wHour>=8 AND NowTimeData.wMinute>=00  AND NowTimeData.wSecond>=00 AND NowDay<>NowTimeData.wDay THEN
		HistoryData_Step:=100;(*8点钟机台断电，错过数据移位。重新移位数据*)
	ELSIF NowTimeData.wHour=8 AND NowTimeData.wMinute=00  AND NowTimeData.wSecond=00 AND NowDay=NowTimeData.wDay THEN
		HistoryData_Step:=100;
	END_IF
100:
(**************************************前一天白班夜班的历史数据移位*************************************************)
	FOR  i :=6 TO 1 BY -1 DO
			DayHistory[i+1]:=DayHistory[i] ;(*日*)
			MonthHistory[i+1]:=MonthHistory[i] ;(*月*)
			HistoryTotal[i+1]:=HistoryTotal[i];(*历史每天生产总数*)
			HistoryOK[i+1]:=HistoryOK[i];(*历史每天生产OK总数*)
			HistoryNG[i+1]:=HistoryNG[i];(*历史每天生产NG总数*)
			HistoryTotal_AM[i+1]:=HistoryTotal_AM[i];(*历史每天白班生产总数*)
			HistoryTotal_PM[i+1]:=HistoryTotal_PM[i];(*历史每天夜班生产总数*)
			HistoryRate_AM[i+1]:=HistoryRate_AM[i];(*历史每天白班良率*)
			HistoryRate_PM[i+1]:=HistoryRate_PM[i];(*历史每天夜班良率*)
			HistoryOK_AM[i+1]:=HistoryOK_AM[i];(*历史每天白班生产OK总数*)
			HistoryOK_PM[i+1]:=HistoryOK_PM[i];(*历史每天夜班生产OK总数*)
			HistoryNG_AM[i+1]:=HistoryNG_AM[i];(*历史每天白班生产NG总数*)
			HistoryNG_PM[i+1]:=HistoryNG_PM[i];(*历史每天夜班生产NG总数*)
			HistoryRun_AM[i+1]:=HistoryRun_AM[i];(*历史每天白班总运行时间合计*)
			HistoryRun_PM[i+1]:=HistoryRun_PM[i];(*历史每天夜班总运行时间合计*)
			HistoryWait_AM[i+1]:=HistoryWait_AM[i];(*历史每天白班总待料时间合计*)
			HistoryWait_PM[i+1]:=HistoryWait_PM[i];(*历史每天夜班总待料时间合计*)
			HistoryAlarm_AM[i+1]:=HistoryAlarm_AM[i];(*历史每天白班总报警时间合计*)
			HistoryAlarm_PM[i+1]:=HistoryAlarm_PM[i];(*历史每天夜班总报警时间合计*)
			
			FOR j := 1 TO 50 DO(*i表示天数，j表示1-10不良分类*)
				HistoryNGClass_AM[i+1,j]:=HistoryNGClass_AM[i,j];(*历史每天白班各类NG数量*)
				HistoryNGClass_PM[i+1,j]:=HistoryNGClass_PM[i,j];(*历史每天夜班各类NG数量*)
				HisTodayNGQualified[i+1,j]:=HisTodayNGQualified[i,j];//历史白班各种NG类型NG率
				HisNightNGQualified[i+1,j]:=HisNightNGQualified[i,j];//历史夜班各种NG类型NG率
			END_FOR
			FOR j := 8 TO 19 DO(*j表示小时*)
				HistoryHour_AM[i+1,j]:=HistoryHour_AM[i,j];(*历史每天白班每小时产量*)
				HistoryRun_AMH[i+1,j]:=HistoryRun_AMH[i,j];(*历史每天白班每小时运行时间合计ARRAY[1..7 ]*)
				HistoryWait_AMH[i+1,j]:=HistoryWait_AMH[i,j];(*历史每天白班每小时待料时间合计ARRAY[1..7 ]*)
				HistoryAlarm_AMH[i+1,j]:=HistoryAlarm_AMH[i,j];(*历史每天白班每小时报警时间合计ARRAY[1..7 ]*)
			END_FOR
			FOR j := 0 TO 23 DO(*j表示小时*)
				HistoryHour_PM[i+1,j]:=HistoryHour_PM [i,j];(*夜班移位每小时产量*)
				HistoryRun_PMH[i+1,j]:=HistoryRun_PMH[i,j];(*历史每天夜班每小时运行时间合计ARRAY[1..7 ]*)
				HistoryWait_PMH[i+1,j]:=HistoryWait_PMH[i,j];(*历史每天夜班每小时待料时间合计ARRAY[1..7 ]*)
				HistoryAlarm_PMH[i+1,j]:=HistoryAlarm_PMH[i,j];(*历史每天夜班每小时报警时间合计ARRAY[1..7 ]*)
			END_FOR
	END_FOR
	HistoryData_Step:=200;
200:
(*******将当天日期和数据传送到历史数据存储区***************)
	DayHistory[1]:= NowDay;
	MonthHistory[1]:=NowMonth;
	HistoryTotal[1]:=TodayTotal;(*历史每天生产总数*)
	HistoryOK[1]:=TodayOK;(*历史每天生产OK总数*)
	HistoryNG[1]:=TodayNG;(*历史每天生产NG总数*)
	HistoryTotal_AM[1]:=TodayTotal_AM;(*历史每天白班生产总数*)
	HistoryTotal_PM[1]:=TodayTotal_PM;(*历史每天夜班生产总数*)
	HistoryRate_AM[1]:=TodayRate_AM;(*历史每天白班良率*)
	HistoryRate_PM[1]:=TodayRate_PM;(*历史每天夜班良率*)
	HistoryOK_AM[1]:=TodayOK_AM;(*历史每天白班生产OK总数*)
	HistoryOK_PM[1]:=TodayOK_PM;(*历史每天夜班生产OK总数*)
	HistoryNG_AM[1]:=TodayNG_AM;(*历史每天白班生产NG总数*)
	HistoryNG_PM[1]:=TodayNG_PM;(*历史每天夜班生产NG总数*)
	HistoryRun_AM	[1]:=TodayRun_AM;(*历史每天白班总运行时间合计*)
	HistoryRun_PM[1]:=TodayRun_PM;(*历史每天夜班总运行时间合计*)
	HistoryWait_AM[1]:=TodayWait_AM;(*历史每天白班总待料时间合计*)
	HistoryWait_PM[1]:=TodayWait_PM;(*历史每天夜班总待料时间合计*)
	HistoryAlarm_AM[1]:=TodayAlarm_AM;(*历史每天白班总报警时间合计*)
	HistoryAlarm_PM[1]:=TodayAlarm_PM;(*历史每天夜班总报警时间合计*)
	FOR j := 1 TO 50 DO(*i表示天数，j表示1-30不良分类*)
		HistoryNGClass_AM[1,j]:=TodayNGClass_AM[j];(*历史每天白班各类NG数量*)
		HistoryNGClass_PM[1,j]:=TodayNGClass_PM[j];(*历史每天夜班各类NG数量*)
		HisTodayNGQualified[1,j]:=TodayNGQualified[j];//历史白班各种NG类型NG率
		HisNightNGQualified[1,j]:=NightNGQualified[j];//历史夜班各种NG类型NG率
	END_FOR
	FOR j := 8 TO 19 DO(*j表示小时*)
		HistoryHour_AM[1,j]:=TodayHour_AM[j];(*历史每天白班每小时产量*)
		HistoryRun_AMH[1,j]:=TodayRun_AMH[j];(*历史每天白班每小时运行时间合计ARRAY[1..7 ]*)
		HistoryWait_AMH[1,j]:=TodayWait_AMH[j];(*历史每天白班每小时待料时间合计ARRAY[1..7 ]*)
		HistoryAlarm_AMH[1,j]:=TodayAlarm_AMH[j];(*历史每天白班每小时报警时间合计ARRAY[1..7 ]*)
	END_FOR
	FOR j := 0 TO 23 DO(*j表示小时*)
		HistoryHour_PM[1,j]:=TodayHour_PM [j];(*夜班移位每小时产量*)
		HistoryRun_PMH[1,j]:=TodayRun_PMH[j];(*历史每天夜班每小时运行时间合计ARRAY[1..7 ]*)
		HistoryWait_PMH[1,j]:=TodayWait_PMH[j];(*历史每天夜班每小时待料时间合计ARRAY[1..7 ]*)
		HistoryAlarm_PMH[1,j]:=TodayAlarm_PMH[j];(*历史每天夜班每小时报警时间合计ARRAY[1..7 ]*)
	END_FOR
	
	FOR j:=0 TO 23 DO
			FOR i:=1 TO 50 DO
					HisTodayNgHour_Day[i,j,1] :=TodayNgHour_Day[i,j];//l历史白班每小时NG类型统计,,
					HisTodayNgHour_Night[i,j,1]:=TodayNgHour_Night[i,j];//历史夜班每小时NG类型统计,,
			END_FOR
	END_FOR
	HistoryData_Step:=300;
300:
(******清除当天数据，并记录当天日期*******)
	NowDay:=NowTimeData.wDay;
	NowMonth:=NowTimeData.wMonth;
	FOR i:=8 TO 19 DO
		TodayHour_AM[i]:=0;(*当天白班每小时产量*)
		RunCnt_AM[i]:=0;		(*白班运行时间计数*)
		WaitCnt_AM[i]:=0;	(*白班待料时间计数*)
		AlarmCnt_AM[i]:=0;	(*白班报警时间计数*)
		TodayRun_AMH[i]:=0;
		TodayWait_AMH[i]:=0;
		TodayAlarm_AMH[i]:=0;
	END_FOR
	FOR i:=0 TO 23 DO
		TodayHour_PM[i]:=0;(*当天夜班每小时产量*)
		RunCnt_PM[i]:=0;		(*夜班运行时间计数*)
		WaitCnt_PM[i]:=0;	(*夜班待料时间计数*)
		AlarmCnt_PM[i]:=0;	(*夜班报警时间计数*)
		TodayRun_PMH[i]:=0;
		TodayWait_PMH[i]:=0;
		TodayAlarm_PMH[i]:=0;
	END_FOR
	FOR i:=1 TO 50 DO
		TodayNGClass_AM[i]:=0;(*当天白班各类NG数量*)
		TodayNGClass_PM[i]:=0;(*当天夜班各类NG数量*)
		TodayNGQualified[i]:=0;//当天白班各种NG类型NG率
		NightNGQualified[i]:=0;//当天夜班各种NG类型NG率	
	END_FOR
	TodayTotal:=0;(*当天生产总数*)
	TodayOK:=0;(*当天生产OK总数*)
	TodayNG:=0;(*当天生产NG总数*)
	TodayTotal_AM:=0;(*当天白班生产总数*)
	TodayTotal_PM:=0;(*当天夜班生产总数*)
	TodayRate_AM:=0;(*当天白班良率*)
	TodayRate_PM:=0;(*当天夜班良率*)
	TodayOK_AM:=0;(*当天白班生产OK总数*)
	TodayOK_PM:=0;(*当天夜班生产OK总数*)
	TodayNG_AM:=0;(*当天白班生产NG总数*)
	TodayNG_PM:=0;(*当天夜班生产NG总数*)
	TodayRun_AM:=0;(*当天白班总运行时间合计*)
	TodayRun_PM:=0;(*当天夜班总运行时间合计*)
	TodayWait_AM:=0;(*当天白班总待料时间合计*)
	TodayWait_PM:=0;(*当天夜班总待料时间合计*)
	TodayAlarm_AM:=0;(*当天白班总报警时间合计*)
	TodayAlarm_PM:=0;(*当天夜班总报警时间合计*)
	FOR i:=1 TO 50 DO
		FOR j:= 0 TO 23 DO
			TodayNgHour_Day[i,j]:=0;//白班每小时NG类型统计,,
			TodayNgHour_Night[i,j]:=0;//夜班每小时NG类型统计,,
		END_FOR
	END_FOR
	SaveDataDelay(IN:=FALSE);
	HistoryData_Step:=400;
400:
	SaveDataDelay(IN:=TRUE,PT:=t#2s, Q=> , ET=> );
	IF SaveDataDelay.Q THEN
		SaveDataDelay(IN:=FALSE);
		HistoryData_Step:=0;
	END_IF
END_CASE
(*************历史数据存储**************)



//	OEE稼动率:=24小时总运行时间/总报警时间+总运行时间
//OEE:=(TodayRun_AM+TodayRun_PM)/((TodayRun_AM+TodayRun_PM)+(TodayAlarm_AM+TodayAlarm_PM));

END_FUNCTION_BLOCK

// ---- POUs/POUs/CaPart.TcPOU
PROGRAM CaPart
VAR_INPUT
          iMode                      :INT;
END_VAR

VAR
	fbCaPart: FB_UserMain;
END_VAR

CALL();
ACT();

ACTION ACT:
(********模切小时、天产能**********)
(*
aCaDay_date(
EE:=Q204[7],
);
*)
//运行时间统计
Catimedata(
	Month:= PLC_wMonth, 
	dDay:=PLC_wDay , 
	Hour:=PLC_wHour , 
	Mins:=PLC_wMinute , 
	Second:=PLC_wSecond , 
	Alm:=stSysState.bErrorStop AND NOT bAnDoorALM AND 
             NOT (ProductPar.CaPar.MQ.bWindSelect AND  ProductPar.parFilterAD[13].Out_Value<=ProductPar.CaPar.fDiameterAlarm_L) AND 
             NOT ( NOT ProductPar.CaPar.MQ.bWindSelect AND  ProductPar.parFilterAD[14].Out_Value<=ProductPar.CaPar.fDiameterAlarm_R) , 
	Wait:=(stSysState.iModehmi=2 OR  stSysState.iModehmi=3 )AND (stSysState.bErrorStop OR bAnDoorALM) AND
             NOT (ProductPar.CaPar.MQ.bWindSelect AND  ProductPar.parFilterAD[13].Out_Value<=ProductPar.CaPar.fDiameterAlarm_L) AND 
             NOT ( NOT ProductPar.CaPar.MQ.bWindSelect AND  ProductPar.parFilterAD[14].Out_Value<=ProductPar.CaPar.fDiameterAlarm_R)   , 
	Run:=stSysState.iModehmi=1  , 
	JP_Wait:=(ProductPar.CaPar.MQ.bWindSelect AND  ProductPar.parFilterAD[13].Out_Value<=ProductPar.CaPar.fDiameterAlarm_L) OR ( NOT ProductPar.CaPar.MQ.bWindSelect AND  ProductPar.parFilterAD[14].Out_Value<=ProductPar.CaPar.fDiameterAlarm_R) , 
	Query:=MQQuery , 
	STTimedata=> , 
	date1:=MQdate );
END_ACTION

ACTION CALL:
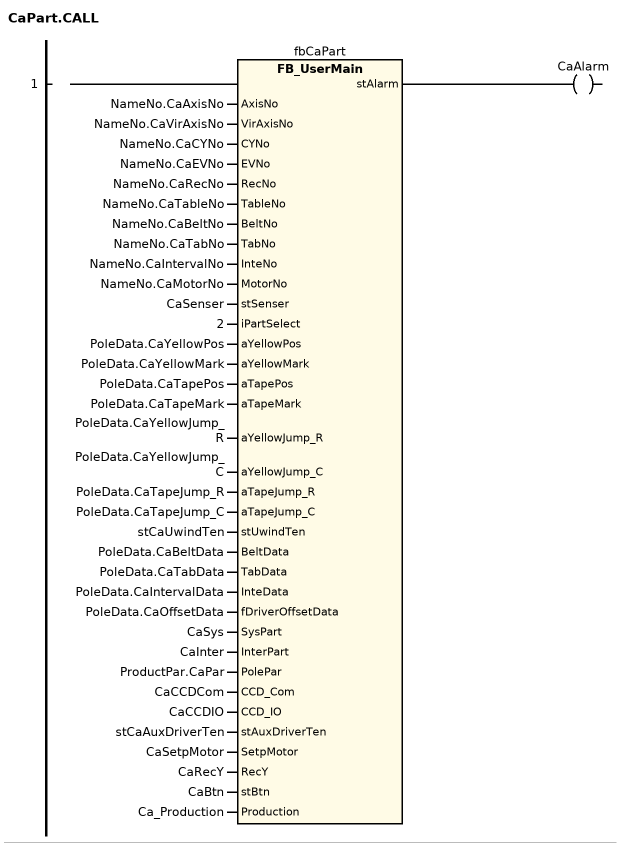
// NETWORK 1
fbCaPart(
    AxisNo := NameNo.CaAxisNo,
    VirAxisNo := NameNo.CaVirAxisNo,
    CYNo := NameNo.CaCYNo,
    EVNo := NameNo.CaEVNo,
    RecNo := NameNo.CaRecNo,
    TableNo := NameNo.CaTableNo,
    BeltNo := NameNo.CaBeltNo,
    TabNo := NameNo.CaTabNo,
    InteNo := NameNo.CaIntervalNo,
    MotorNo := NameNo.CaMotorNo,
    stSenser := CaSenser,
    iPartSelect := 2,
    aYellowPos := PoleData.CaYellowPos,
    aYellowMark := PoleData.CaYellowMark,
    aTapePos := PoleData.CaTapePos,
    aTapeMark := PoleData.CaTapeMark,
    aYellowJump_R := PoleData.CaYellowJump_R,
    aYellowJump_C := PoleData.CaYellowJump_C,
    aTapeJump_R := PoleData.CaTapeJump_R,
    aTapeJump_C := PoleData.CaTapeJump_C,
    stUwindTen := stCaUwindTen,
    BeltData := PoleData.CaBeltData,
    TabData := PoleData.CaTabData,
    InteData := PoleData.CaIntervalData,
    fDriverOffsetData := PoleData.CaOffsetData,
    SysPart := CaSys,
    InterPart := CaInter,
    PolePar := ProductPar.CaPar,
    CCD_Com := CaCCDCom,
    CCD_IO := CaCCDIO,
    stAuxDriverTen := stCaAuxDriverTen,
    SetpMotor := CaSetpMotor,
    RecY := CaRecY,
    stBtn := CaBtn,
    Production := Ca_Production); // FB_UserMain
CaAlarm := fbCaPart.stAlarm;
END_ACTION

END_PROGRAM

// ---- POUs/BasicFunction/Data/FC_Variance.TcPOU
FUNCTION FC_Variance : REAL
VAR_INPUT
a: ARRAY [1..10] OF REAL;
END_VAR
VAR
b:REAL;
test:BOOL;
ii1:INT;
c:REAL;
d:real;
END_VAR

test:=FALSE;
FOR ii1:=1 TO 10 BY 1 DO
	IF a[ii1]=0 THEN
		test:=TRUE;
	END_IF
END_FOR
IF test THEN
	FC_Variance:=0;
ELSE
	b:=0;
	//FOR ii1:=1 TO 10 BY 1 DO
	//	b:=b+a[ii1];
	//END_FOR	
	c:=b/10;	
	d:=0;
	FOR ii1:=1 TO 10 BY 1 DO
		d:=d+(c-a[ii1])*(c-a[ii1]);
	END_FOR
	FC_Variance:=d/10;
END_IF

END_FUNCTION

// ---- POUs/POUs/FingerprintKey.TcPOU
PROGRAM FingerprintKey
VAR
	AnID: STRING(49);
	CaID: STRING(49);
	AnLevel: STRING(49);
	CaLevel: STRING(49);
	AnLoginSuccess: BOOL;//正极指纹匹配成功
	CaLoginSuccess: BOOL;//负极指纹匹配成功
	Keyton:  ARRAY[0..10] OF TON;//1:获取用户及权限延时
	AnLevelHMI_Read: BYTE;//触摸屏权限，用于触摸屏读取用户索引
	CaLevelHMI_Read: BYTE;//触摸屏权限，用于触摸屏读取用户索引
	AnPassWord: STRING(16);//触摸屏密码，用于触摸屏读取用户对应密码
	CaPassWord: STRING(16);//触摸屏密码，用于触摸屏读取用户对应密码
	AnLevelHMI_Write: INT;//触摸屏权限，用于触摸屏反馈给PLC
	CaLevelHMI_Write: INT;//触摸屏权限，用于触摸屏反馈给PLC
	AnKeyStep: INT;//正极权限判断自动
	CaKeyStep: INT;//正极权限判断自动
	Anblogin: BOOL;
	Cablogin: BOOL;
END_VAR

//正极模切变量（指纹机1）
User01.AnMQ_FingerprintKey.MachineId ;//指纹器编号
User01.AnMQ_FingerprintKey.UserId;//用户名
User01.AnMQ_FingerprintKey.UserClassLevel;//用户权限
User01.AnMQ_FingerprintKey.Fid;//本地文件id
User01.AnMQ_FingerprintKey.MatchScore;//指纹匹配评分
User01.AnMQ_FingerprintKey.Result;//匹配结果
User01.AnMQ_FingerprintKey.FileName;//本地文件路径



////////////////////////////////////////////////////////////////////////正极指纹仪自动程序///////////////////////////////////////////////////////////////
Keyton[1](IN:=AnLoginSuccess , PT:=T#100MS , Q=> , ET=> );

IF User01.AnMQ_FingerprintKey.MachineId='01' THEN
	IF User01.AnMQ_FingerprintKey.Result='Success' THEN
		AnLoginSuccess:=TRUE;//指纹匹配成功
	END_IF	
END_IF


CASE AnKeyStep OF
0:
	IF Keyton[1].Q THEN
		IF User01.AnMQ_FingerprintKey.UserId<>'' AND User01.AnMQ_FingerprintKey.UserClassLevel<>'' THEN
			AnID:=User01.AnMQ_FingerprintKey.UserId;
			AnLevel:=User01.AnMQ_FingerprintKey.UserClassLevel;
			AnLevelHMI_Read:=0;
			IF AnID=User01.AnMQ_FingerprintKey.UserId AND AnLevel=User01.AnMQ_FingerprintKey.UserClassLevel THEN
				AnKeyStep:=100;
			END_IF
		END_IF
	END_IF
100://用户权限判断	(触摸屏读取时，采用用户索引，顺序要与触摸屏用户顺序一致）
	IF AnLevel='PRD' THEN
		AnLevelHMI_Read:=1;
		//PassWord:='1111';
		IF AnLevelHMI_Read=1  THEN//AND PassWord='1111'
			AnKeyStep:=200;
		END_IF
	ELSIF AnLevel='ME' THEN
		AnLevelHMI_Read:=2;
		//PassWord:='SWD123';
		IF AnLevelHMI_Read=2  THEN//AND PassWord='SWD123'
			AnKeyStep:=200;
		END_IF
	ELSIF AnLevel='PRJ' THEN
		AnLevelHMI_Read:=3;
		//PassWord:='SWDQDJ';
		IF AnLevelHMI_Read=3  THEN//AND PassWord='SWDQDJ'
			AnKeyStep:=200;
		END_IF
	ELSIF AnLevel='GYS' THEN
		AnLevelHMI_Read:=4;
		//PassWord:='YK556';
		IF AnLevelHMI_Read=4 THEN// AND PassWord='YK556'
			AnKeyStep:=200;
		END_IF
	ELSIF AnLevel='QA' THEN
		AnLevelHMI_Read:=5;
		//PassWord:='OYX98766';
		IF AnLevelHMI_Read=5  THEN//AND PassWord='OYX98766'
			AnKeyStep:=200;
		END_IF
	ELSIF AnLevel='KF' THEN
		AnLevelHMI_Read:=6;
		//PassWord:='0513';
		IF AnLevelHMI_Read=6  THEN//AND PassWord='0513'
			AnKeyStep:=200;
		END_IF
	ELSIF AnLevel='Safe' THEN
		AnLevelHMI_Read:=7;
		//PassWord:='87558';
		IF AnLevelHMI_Read=7 THEN//AND PassWord='87558'
			AnKeyStep:=200;
		END_IF
	ELSE
		AnLoginSuccess:=FALSE;
		AnLevel:='';
		User01.AnMQ_FingerprintKey.Result:='';
		User01.AnMQ_FingerprintKey.UserId:='';
		User01.AnMQ_FingerprintKey.UserClassLevel:='';
		User01.AnMQ_FingerprintKey.MachineId:='';
		AnKeyStep:=0;
	END_IF
	
200:
		Anblogin:=TRUE;
		AnLoginSuccess:=FALSE;
		AnKeyStep:=300;

300:
		IF AnLevelHMI_Write=1 THEN
		AnLevelHMI_Read:=0;
		AnPassWord:='';
		AnLoginSuccess:=FALSE;
		AnLevel:='';
		User01.AnMQ_FingerprintKey.Result:='';
		User01.AnMQ_FingerprintKey.UserId:='';
		User01.AnMQ_FingerprintKey.UserClassLevel:='';
		User01.AnMQ_FingerprintKey.MachineId:='';
		AnKeyStep:=0;
		Anblogin:=FALSE;
		AnLoginSuccess:=FALSE;
		AnLevelHMI_Write:=0;
		END_IF
END_CASE



//负极模切变量（指纹机2）
User01.CaMQ_FingerprintKey.MachineId ;//指纹器编号
User01.CaMQ_FingerprintKey.UserId;//用户名
User01.CaMQ_FingerprintKey.UserClassLevel;//用户权限
User01.CaMQ_FingerprintKey.Fid;//本地文件id
User01.CaMQ_FingerprintKey.MatchScore;//指纹匹配评分
User01.CaMQ_FingerprintKey.Result;//匹配结果
User01.CaMQ_FingerprintKey.FileName;//本地文件路径


///////////////////////////////////////////////////////////////////////////负极指纹仪自动程序/////////////////////////////////////////////////////////////////////
Keyton[2](IN:=CaLoginSuccess , PT:=T#100MS , Q=> , ET=> );

IF User01.CaMQ_FingerprintKey.MachineId='02' THEN
	IF User01.CaMQ_FingerprintKey.Result='Success' THEN
		CaLoginSuccess:=TRUE;//指纹匹配成功
	END_IF	
END_IF


CASE CaKeyStep OF
0:
	IF Keyton[2].Q THEN
		IF User01.CaMQ_FingerprintKey.UserId<>'' AND User01.CaMQ_FingerprintKey.UserClassLevel<>'' THEN
			CaID:=User01.CaMQ_FingerprintKey.UserId;
			CaLevel:=User01.CaMQ_FingerprintKey.UserClassLevel;
			CaLevelHMI_Read:=0;
			IF CaID=User01.CaMQ_FingerprintKey.UserId AND CaLevel=User01.CaMQ_FingerprintKey.UserClassLevel THEN
				CaKeyStep:=100;
			END_IF
		END_IF
	END_IF
100://用户权限判断	(触摸屏读取时，采用用户索引，顺序要与触摸屏用户顺序一致）
	IF CaLevel='PRD' THEN
		CaLevelHMI_Read:=1;
		//PassWord:='1111';
		IF CaLevelHMI_Read=1  THEN//AND PassWord='1111'
			CaKeyStep:=200;
		END_IF
	ELSIF CaLevel='ME' THEN
		CaLevelHMI_Read:=2;
		//PassWord:='SWD123';
		IF CaLevelHMI_Read=2  THEN//AND PassWord='SWD123'
			CaKeyStep:=200;
		END_IF
	ELSIF CaLevel='PRJ' THEN
		CaLevelHMI_Read:=3;
		//PassWord:='SWDQDJ';
		IF CaLevelHMI_Read=3  THEN//AND PassWord='SWDQDJ'
			CaKeyStep:=200;
		END_IF
	ELSIF CaLevel='GYS' THEN
		CaLevelHMI_Read:=4;
		//PassWord:='YK556';
		IF CaLevelHMI_Read=4 THEN// AND PassWord='YK556'
			CaKeyStep:=200;
		END_IF
	ELSIF CaLevel='QA' THEN
		CaLevelHMI_Read:=5;
		//PassWord:='OYX98766';
		IF CaLevelHMI_Read=5  THEN//AND PassWord='OYX98766'
			CaKeyStep:=200;
		END_IF
	ELSIF CaLevel='KF' THEN
		CaLevelHMI_Read:=6;
		//PassWord:='0513';
		IF CaLevelHMI_Read=6  THEN//AND PassWord='0513'
			CaKeyStep:=200;
		END_IF
	ELSIF CaLevel='Safe' THEN
		CaLevelHMI_Read:=7;
		//PassWord:='87558';
		IF CaLevelHMI_Read=7 THEN//AND PassWord='87558'
			CaKeyStep:=200;
		END_IF
	ELSE
		CaLoginSuccess:=FALSE;
		CaLevel:='';
		User01.CaMQ_FingerprintKey.Result:='';
		User01.CaMQ_FingerprintKey.UserId:='';
		User01.CaMQ_FingerprintKey.UserClassLevel:='';
		User01.CaMQ_FingerprintKey.MachineId:='';
		CaKeyStep:=0;
	END_IF
	
200:
		Cablogin:=TRUE;
		CaLoginSuccess:=FALSE;
		CaKeyStep:=300;
300:
	IF CaLevelHMI_Write=1 THEN
		CaLevelHMI_Read:=0;
		CaPassWord:='';
		CaLoginSuccess:=FALSE;
		CaLevel:='';
		User01.CaMQ_FingerprintKey.Result:='';
		User01.CaMQ_FingerprintKey.UserId:='';
		User01.CaMQ_FingerprintKey.UserClassLevel:='';
		User01.CaMQ_FingerprintKey.MachineId:='';
		CaLevelHMI_Write:=0;
		CaKeyStep:=0;
	END_IF
END_CASE

END_PROGRAM

// ---- POUs/BasicFunction/SystemInfo/SystemInfoCtrl.TcPOU
FUNCTION_BLOCK SystemInfoCtrl
VAR_INPUT
	Reset					: BOOL;
	RTCSyncCylce		:	DWORD := 5; (* in seconds *)
	TimeStampTrig		:	BOOL;
END_VAR
VAR_OUTPUT
//	RunTimeNo			: BYTE;
//	ProjectName			: STRING(32);
//	NumberOfTasks		: BYTE;
//	OnlineChangeCount	: UINT;
	RetainVarErr		: BOOL;
	PersistenVarErr	: BOOL;
	TimeStampDT			:	DATE_AND_TIME;
	TimeStamp			:	STRING(25); (* DD.MM.YY-Stunde:Minute:Sekunde:xxx *)
	TimeStr				:	STRING(15);	(* hh.mm.ss.xxms *)
	DateStr				:	STRING(15);	(* dd.mm.jj *)
	TimeStamp2			:	STRING(25); (* YYYY-MM-DD_HHMMSS for example YYYY-MM-DD_HHMMSS_Name.txt *)
	TimeStruct			:	TIMESTRUCT;
	MonthDays			:	WORD;
	LeapYear				:	BOOL;
	WeekOfYear			:	WORD;
	timezoneId			: 	E_TimeZoneID;
END_VAR

VAR
	(* Inst. Get Taskindex *)
	InstGETCURTASKINDEX	: 	GETCURTASKINDEX;
	InstLocalSystemTime	:	FB_LocalSystemTime;

	(* Info: SystemInfo.bootDataFlags
	Bit
	0 RETAIN Variablen: LOADED (fehlerfrei geladen)
	1 RETAIN Variablen: INVALID (es wurde die Sicherungskopie geladen, weil keine g黮tige Datei vorhanden war)
	2 RETAIN Variablen: REQUESTED (RETAIN Variablen sollten geladen werden, Einstellung im TwinCAT System Control))
	3 reserviert
	4 PERSISTENT Variablen: LOADED (fehlerfrei geladen)
	5 PERSISTENT Variablen: INVALID (es wurde die Sicherungskopie geladen, weil keine g黮tige Datei vorhanden war)
	6 reserviert
	7 reserviert *)

	RetainVarLoaded			: BOOL;
	RetainVarInvalid		: BOOL;
	RetainVarRequested		: BOOL;
	PersistentVarLoaded		: BOOL;
	PersistentVarInvalid	: BOOL;

	(* Info: SystemTaskInfoArr	(* Ist ein Array von 1-4 *)
	active					:	BOOL; 		(* Diese Variable zeigt an, ob die Task aktiv ist.*)
	taskName					:	STRING(16);	(* Der Taskname.*)
	firstCycle				:	BOOL;			(* Diese Variable hat im ersten Zyklus der SPS-Task den Wert: TRUE.*)
	cycleTimeExceeded		:	BOOL;			(* In dieser Variablen wird ein 躡erschreiten der eingestellten Taskzykluszeit gemeldet*)
	cycleTime				:	UDINT;		(* Eingestellte Taskzykluszeit in Vielfachen von 100ns*)
	lastExecTime			:	UDINT;		(* Ben鰐igte Zykluszeit f黵 den letzten Zyklus in Vielfachen von 100 ns*)
	priority					:	BYTE;			(* Eingestellte Prioritaet der Task*)
	cycleCount				: 	UDINT;		(* Zykluszaehler*) *)
	_sec						:	WORD;
//	_hour						:	WORD;
END_VAR

(* Get Current Task Index ************************************************************************)
	InstGETCURTASKINDEX();

(* Read System Info Current Task *****************************************************************)
	(* Task Info *)
//	RunTimeNo				:=  _AppInfo.runTimeNo;
//	ProjectName				:=  _AppInfo.ProjectName;
//	NumberOfTasks 			:=  _AppInfo.TaskCnt;
//	OnlineChangeCount		:=  _AppInfo.OnlineChangeCnt;

	(* System Boot Flags *)
//	RetainVarLoaded		:= SystemInfo.bootDataFlags.0;
//	RetainVarInvalid		:= SystemInfo.bootDataFlags.1 ;
//	RetainVarRequested 	:= SystemInfo.bootDataFlags.2 ;
//	PersistentVarLoaded	:= SystemInfo.bootDataFlags.4;
//	PersistentVarInvalid	:= SystemInfo.bootDataFlags.5;


	(* Retein/Persisten Data Err *)
	IF  _TaskInfo[InstGETCURTASKINDEX.Index].FirstCycle THEN
		RetainVarErr		:= NOT RetainVarLoaded AND RetainVarRequested OR RetainVarInvalid;
		PersistenVarErr	:= NOT PersistentVarLoaded OR PersistentVarInvalid;
	ELSIF Reset THEN
		M_Reset();
	ELSE
		;
	END_IF

(* Systemzeit auslesen ************************************************************************)
	InstLocalSystemTime(
		sNetID		:= '',
		bEnable		:= TRUE,
		dwCycle		:= RTCSyncCylce,
		dwOpt			:= (* Default *),
		tTimeout		:= (* Default *),
		bValid		=> ,
		systemTime	=> TimeStruct,
		tzID			=> timezoneId);

	IF TimeStampTrig
		AND InstLocalSystemTime.bValid
	THEN
		(* Date dd.mm.jj ********************)
		IF TimeStruct.wDay < 10 THEN
			DateStr := CONCAT('0',WORD_TO_STRING(TimeStruct.wDay));
		ELSE
			DateStr := WORD_TO_STRING(TimeStruct.wDay);
		END_IF
		DateStr := CONCAT(DateStr,'.');
		IF TimeStruct.wMonth < 10 THEN
			DateStr := CONCAT(DateStr,CONCAT('0',WORD_TO_STRING(TimeStruct.wMonth)));
		ELSE
			DateStr := CONCAT(DateStr,WORD_TO_STRING(TimeStruct.wMonth));
		END_IF
		DateStr := CONCAT(DateStr,'.');
		DateStr := CONCAT(DateStr,RIGHT(WORD_TO_STRING(TimeStruct.wYear),2));
	
		(* Time hh.mm.ss.xxms ***************)
		IF TimeStruct.wHour < 10 THEN
			TimeStr := CONCAT('0',WORD_TO_STRING(TimeStruct.wHour));
		ELSE
			TimeStr := WORD_TO_STRING(TimeStruct.wHour);
		END_IF
		TimeStr := CONCAT(TimeStr,':');
		IF TimeStruct.wMinute < 10 THEN
			TimeStr := CONCAT(TimeStr,CONCAT('0',WORD_TO_STRING(TimeStruct.wMinute)));
		ELSE
			TimeStr := CONCAT(TimeStr,WORD_TO_STRING(TimeStruct.wMinute));
		END_IF
		TimeStr := CONCAT(TimeStr,':');
		IF TimeStruct.wSecond < 10 THEN
			TimeStr := CONCAT(TimeStr,CONCAT('0',WORD_TO_STRING(TimeStruct.wSecond)));
		ELSE
			TimeStr := CONCAT(TimeStr,WORD_TO_STRING(TimeStruct.wSecond));
		END_IF
	
		(* TimeStamp Format DE: DD.MM.YY-Stunde:Minute:Sekunde:xxx,*)
		TimeStamp := CONCAT(DateStr,'-');
		TimeStamp := CONCAT(TimeStamp,TimeStr);
		TimeStamp := CONCAT(TimeStamp,':');
		IF TimeStruct.wMilliseconds > 100 THEN
			TimeStamp:=CONCAT(TimeStamp,WORD_TO_STRING(TimeStruct.wMilliseconds));
		ELSIF TimeStruct.wMilliseconds > 10 THEN
			TimeStamp:=CONCAT(CONCAT(TimeStamp,'0'),WORD_TO_STRING(TimeStruct.wMilliseconds));
		ELSE
			TimeStamp:=CONCAT(CONCAT(TimeStamp,'00'),WORD_TO_STRING(TimeStruct.wMilliseconds));
		END_IF
	
		(* Timestamp Format ENG: YYYY-MM-DD-hh:mm:ss.xxx *)
		(* TimeStamp := SYSTEMTIME_TO_STRING(TimeStruct); *)
	
		(* TimeStamp2 FileName YYYY-MM-DD_HHMMSS *)
		IF _sec <> TimeStruct.wSecond THEN
			TimeStamp2 := CONCAT(WORD_TO_STRING(TimeStruct.wYear),'-');
			IF TimeStruct.wMonth < 10 THEN
				TimeStamp2 := CONCAT(TimeStamp2,CONCAT('0',WORD_TO_STRING(TimeStruct.wMonth)));
			ELSE
				TimeStamp2 := CONCAT(TimeStamp2,WORD_TO_STRING(TimeStruct.wMonth));
			END_IF
			TimeStamp2 := CONCAT(TimeStamp2,'-');
			IF TimeStruct.wDay < 10 THEN
				TimeStamp2 := CONCAT(TimeStamp2,CONCAT('0',WORD_TO_STRING(TimeStruct.wDay)));
			ELSE
				TimeStamp2 := CONCAT(TimeStamp2,WORD_TO_STRING(TimeStruct.wDay));
			END_IF
			TimeStamp2 := CONCAT(TimeStamp2,'_');
			IF TimeStruct.wHour < 10 THEN
				TimeStamp2 := CONCAT(TimeStamp2,CONCAT('0',WORD_TO_STRING(TimeStruct.wHour)));
			ELSE
				TimeStamp2 := CONCAT(TimeStamp2,WORD_TO_STRING(TimeStruct.wHour));
			END_IF
			IF TimeStruct.wMinute < 10 THEN
				TimeStamp2 := CONCAT(TimeStamp2,CONCAT('0',WORD_TO_STRING(TimeStruct.wMinute)));
			ELSE
				TimeStamp2 := CONCAT(TimeStamp2,WORD_TO_STRING(TimeStruct.wMinute));
			END_IF
			IF TimeStruct.wSecond < 10 THEN
				TimeStamp2 := CONCAT(TimeStamp2,CONCAT('0',WORD_TO_STRING(TimeStruct.wSecond)));
			ELSE
				TimeStamp2 := CONCAT(TimeStamp2,WORD_TO_STRING(TimeStruct.wSecond));
			END_IF
			_sec := TimeStruct.wSecond;
	
			(* Jahresinformationen *)
			TimeStampDT := SYSTEMTIME_TO_DT(TimeStruct);
			MonthDays	:= F_GetMaxMonthDays(TimeStruct.wYear,TimeStruct.wMonth);
			LeapYear		:= F_YearIsLeapYear(TimeStruct.wYear) ;
			WeekOfYear	:= F_GetWeekOfTheYear(TimeStampDT);
	
		END_IF
	END_IF

(**************************************************************************************************)

ACTION M_Reset:
RetainVarErr := PersistenVarErr := FALSE;
END_ACTION

END_FUNCTION_BLOCK

// ---- POUs/POUs/ProductLocal.TcPOU
FUNCTION_BLOCK ProductLocal
VAR_INPUT
	NGFlag1:BOOL;(*NG1计数标志*)
	NGFlag2:BOOL;(*NG2计数标志*)
	NGFlag3:BOOL;(*NG3计数标志*)
	NGFlag4:BOOL;(*NG4计数标志*)
	NGFlag5:BOOL;(*NG5计数标志*)
	NGFlag6:BOOL;(*NG6计数标志*)
	NGFlag7:BOOL;(*NG7计数标志*)
	NGFlag8:BOOL;(*NG8计数标志*)
	NGFlag9:BOOL;(*NG9计数标志*)
	NGFlag10:BOOL;(*NG10计数标志*)
	NGFlag11:BOOL;(*NG11计数标志*)
	NGFlag12:BOOL;(*NG12计数标志*)
	NGFlag13:BOOL;(*NG13计数标志*)
	NGFlag14:BOOL;(*NG14计数标志*)
	NGFlag15:BOOL;(*NG15计数标志*)
	NGFlag16:BOOL;(*NG16计数标志*)
	NGFlag17:BOOL;(*NG17计数标志*)
	NGFlag18:BOOL;(*NG18计数标志*)
	NGFlag19:BOOL;(*NG19计数标志*)
	NGFlag20:BOOL;(*NG20计数标志*)
	NGFlag21:BOOL;(*NG21计数标志*)
	NGFlag22:BOOL;(*NG22计数标志*)
	NGFlag23:BOOL;(*NG23计数标志*)
	NGFlag24:BOOL;(*NG24计数标志*)
	NGFlag25:BOOL;(*NG25计数标志*)
	NGFlag26:BOOL;(*NG26计数标志*)
	NGFlag27:BOOL;(*NG27计数标志*)
	NGFlag28:BOOL;(*NG28计数标志*)
	NGFlag29:BOOL;(*NG29计数标志*)
	NGFlag30:BOOL;(*NG30计数标志*)
END_VAR
VAR_IN_OUT

END_VAR

VAR_OUTPUT
	TodayNGClass_AM		:ARRAY[1..30 ] 	OF REAL;(*当天白班各类NG数量ARRAY[1..30 ]*)
	TodayNGClass_PM		:ARRAY[1..30 ] 	OF REAL;(*当天夜班各类NG数量ARRAY[1..30 ]*)
	TodayNG_AM:REAL;(*当天白班生产NG总数*)
	TodayNG_PM:REAL;(*当天夜班生产NG总数*)
END_VAR

VAR
	Data_Step:UINT;
	i:UINT;
	TrigNgAdd: ARRAY[1..30 ] OF R_TRIG;(*1-30类ng计数统计*)
	SaveDataDelay:TON;
END_VAR

TrigNgAdd[1](CLK:=NGFlag1,Q=> );(*1类ng*)
TrigNgAdd[2](CLK:=NGFlag2,Q=> );(*2类ng*)
TrigNgAdd[3](CLK:=NGFlag3,Q=> );(*3类ng*)
TrigNgAdd[4](CLK:=NGFlag4,Q=> );(*4类ng*)
TrigNgAdd[5](CLK:=NGFlag5,Q=> );(*5类ng*)
TrigNgAdd[6](CLK:=NGFlag6,Q=> );(*6类ng*)
TrigNgAdd[7](CLK:=NGFlag7,Q=> );(*7类ng*)
TrigNgAdd[8](CLK:=NGFlag8,Q=> );(*8类ng*)
TrigNgAdd[9](CLK:=NGFlag9,Q=> );(*9类ng*)
TrigNgAdd[10](CLK:=NGFlag10,Q=> );(*10类ng*)
TrigNgAdd[11](CLK:=NGFlag11,Q=> );(*11类ng*)
TrigNgAdd[12](CLK:=NGFlag12,Q=> );(*12类ng*)
TrigNgAdd[13](CLK:=NGFlag13,Q=> );(*13类ng*)
TrigNgAdd[14](CLK:=NGFlag14,Q=> );(*14类ng*)
TrigNgAdd[15](CLK:=NGFlag15,Q=> );(*15类ng*)
TrigNgAdd[16](CLK:=NGFlag16,Q=> );(*16类ng*)
TrigNgAdd[17](CLK:=NGFlag17,Q=> );(*17类ng*)
TrigNgAdd[18](CLK:=NGFlag18,Q=> );(*18类ng*)
TrigNgAdd[19](CLK:=NGFlag19,Q=> );(*19类ng*)
TrigNgAdd[20](CLK:=NGFlag20,Q=> );(*20类ng*)
TrigNgAdd[21](CLK:=NGFlag21,Q=> );(*21类ng*)
TrigNgAdd[22](CLK:=NGFlag22,Q=> );(*22类ng*)
TrigNgAdd[23](CLK:=NGFlag23,Q=> );(*23类ng*)
TrigNgAdd[24](CLK:=NGFlag24,Q=> );(*24类ng*)
TrigNgAdd[25](CLK:=NGFlag25,Q=> );(*25类ng*)
TrigNgAdd[26](CLK:=NGFlag26,Q=> );(*26类ng*)
TrigNgAdd[27](CLK:=NGFlag27,Q=> );(*27类ng*)
TrigNgAdd[28](CLK:=NGFlag28,Q=> );(*28类ng*)
TrigNgAdd[29](CLK:=NGFlag29,Q=> );(*29类ng*)
TrigNgAdd[30](CLK:=NGFlag30,Q=> );(*30类ng*)

(***白班数据统计******)
//FOR i:=8 TO 19 DO
	//IF PLC_wHour=i THEN
		IF PLC_wHour>=8 AND PLC_wHour<=19 THEN
			(*******白班NG不良分类统计*)
			IF TrigNgAdd[1].Q THEN
				TodayNGClass_AM[1]:=TodayNGClass_AM[1]+1;
			END_IF
			IF TrigNgAdd[2].Q THEN
				TodayNGClass_AM[2]:=TodayNGClass_AM[2]+1;
			END_IF
			IF TrigNgAdd[3].Q THEN
				TodayNGClass_AM[3]:=TodayNGClass_AM[3]+1;
			END_IF
			IF TrigNgAdd[4].Q THEN
				TodayNGClass_AM[4]:=TodayNGClass_AM[4]+1;
			END_IF
			IF TrigNgAdd[5].Q THEN
				TodayNGClass_AM[5]:=TodayNGClass_AM[5]+1;
			END_IF
			IF TrigNgAdd[6].Q THEN
				TodayNGClass_AM[6]:=TodayNGClass_AM[6]+1;
			END_IF
			IF TrigNgAdd[7].Q THEN
				TodayNGClass_AM[7]:=TodayNGClass_AM[7]+1;
			END_IF
			IF TrigNgAdd[8].Q THEN
				TodayNGClass_AM[8]:=TodayNGClass_AM[8]+1;
			END_IF
			IF TrigNgAdd[9].Q THEN
				TodayNGClass_AM[9]:=TodayNGClass_AM[9]+1;
			END_IF
			IF TrigNgAdd[10].Q THEN
				TodayNGClass_AM[10]:=TodayNGClass_AM[10]+1;
			END_IF
			IF TrigNgAdd[11].Q THEN
				TodayNGClass_AM[11]:=TodayNGClass_AM[11]+1;
			END_IF
			IF TrigNgAdd[12].Q THEN
				TodayNGClass_AM[12]:=TodayNGClass_AM[12]+1;
			END_IF
			IF TrigNgAdd[13].Q THEN
				TodayNGClass_AM[13]:=TodayNGClass_AM[13]+1;
			END_IF
			IF TrigNgAdd[14].Q THEN
				TodayNGClass_AM[14]:=TodayNGClass_AM[14]+1;
			END_IF
			IF TrigNgAdd[15].Q THEN
				TodayNGClass_AM[15]:=TodayNGClass_AM[15]+1;
			END_IF
			IF TrigNgAdd[16].Q THEN
				TodayNGClass_AM[16]:=TodayNGClass_AM[16]+1;
			END_IF
			IF TrigNgAdd[17].Q THEN
				TodayNGClass_AM[17]:=TodayNGClass_AM[17]+1;
			END_IF
			IF TrigNgAdd[18].Q THEN
				TodayNGClass_AM[18]:=TodayNGClass_AM[18]+1;
			END_IF
			IF TrigNgAdd[19].Q THEN
				TodayNGClass_AM[19]:=TodayNGClass_AM[19]+1;
			END_IF
			IF TrigNgAdd[20].Q THEN
				TodayNGClass_AM[20]:=TodayNGClass_AM[20]+1;
			END_IF
			IF TrigNgAdd[21].Q THEN
				TodayNGClass_AM[21]:=TodayNGClass_AM[21]+1;
			END_IF
			IF TrigNgAdd[22].Q THEN
				TodayNGClass_AM[22]:=TodayNGClass_AM[22]+1;
			END_IF
			IF TrigNgAdd[23].Q THEN
				TodayNGClass_AM[23]:=TodayNGClass_AM[23]+1;
			END_IF
			IF TrigNgAdd[24].Q THEN
				TodayNGClass_AM[24]:=TodayNGClass_AM[24]+1;
			END_IF
			IF TrigNgAdd[25].Q THEN
				TodayNGClass_AM[25]:=TodayNGClass_AM[25]+1;
			END_IF
			IF TrigNgAdd[26].Q THEN
				TodayNGClass_AM[26]:=TodayNGClass_AM[26]+1;
			END_IF
			IF TrigNgAdd[27].Q THEN
				TodayNGClass_AM[27]:=TodayNGClass_AM[27]+1;
			END_IF
			IF TrigNgAdd[28].Q THEN
				TodayNGClass_AM[28]:=TodayNGClass_AM[28]+1;
			END_IF
			IF TrigNgAdd[29].Q THEN
				TodayNGClass_AM[29]:=TodayNGClass_AM[29]+1;
			END_IF
			IF TrigNgAdd[30].Q THEN
				TodayNGClass_AM[30]:=TodayNGClass_AM[30]+1;
			END_IF
		END_IF
	//END_IF
//END_FOR

(*当天白班生产NG总数*)
TodayNG_AM:=TodayNGClass_AM[1]+TodayNGClass_AM[2]+TodayNGClass_AM[3]+TodayNGClass_AM[4]+TodayNGClass_AM[5]+
				TodayNGClass_AM[6]+TodayNGClass_AM[7]+TodayNGClass_AM[8]+TodayNGClass_AM[9]+TodayNGClass_AM[10]+
				TodayNGClass_AM[11]+TodayNGClass_AM[12]+TodayNGClass_AM[13]+TodayNGClass_AM[14]+TodayNGClass_AM[15]+
				TodayNGClass_AM[16]+TodayNGClass_AM[17]+TodayNGClass_AM[18]+TodayNGClass_AM[19]+TodayNGClass_AM[20]+
				TodayNGClass_AM[21]+TodayNGClass_AM[22]+TodayNGClass_AM[23]+TodayNGClass_AM[24]+TodayNGClass_AM[25]+
				TodayNGClass_AM[26]+TodayNGClass_AM[27]+TodayNGClass_AM[28]+TodayNGClass_AM[29]+TodayNGClass_AM[30];


(*******夜班数据统计******)
//FOR i:=0 TO 23 DO
	//IF PLC_wHour=i THEN
		IF PLC_wHour<=7 OR PLC_wHour>=20 THEN
			(*******白班NG不良分类统计*)
			IF TrigNgAdd[1].Q THEN
				TodayNGClass_PM[1]:=TodayNGClass_PM[1]+1;
			END_IF
			IF TrigNgAdd[2].Q THEN
				TodayNGClass_PM[2]:=TodayNGClass_PM[2]+1;
			END_IF
			IF TrigNgAdd[3].Q THEN
				TodayNGClass_PM[3]:=TodayNGClass_PM[3]+1;
			END_IF
			IF TrigNgAdd[4].Q THEN
				TodayNGClass_PM[4]:=TodayNGClass_PM[4]+1;
			END_IF
			IF TrigNgAdd[5].Q THEN
				TodayNGClass_PM[5]:=TodayNGClass_PM[5]+1;
			END_IF
			IF TrigNgAdd[6].Q THEN
				TodayNGClass_PM[6]:=TodayNGClass_PM[6]+1;
			END_IF
			IF TrigNgAdd[7].Q THEN
				TodayNGClass_PM[7]:=TodayNGClass_PM[7]+1;
			END_IF
			IF TrigNgAdd[8].Q THEN
				TodayNGClass_PM[8]:=TodayNGClass_PM[8]+1;
			END_IF
			IF TrigNgAdd[9].Q THEN
				TodayNGClass_PM[9]:=TodayNGClass_PM[9]+1;
			END_IF
			IF TrigNgAdd[10].Q THEN
				TodayNGClass_PM[10]:=TodayNGClass_PM[10]+1;
			END_IF
			IF TrigNgAdd[11].Q THEN
				TodayNGClass_PM[11]:=TodayNGClass_PM[11]+1;
			END_IF
			IF TrigNgAdd[12].Q THEN
				TodayNGClass_PM[12]:=TodayNGClass_PM[12]+1;
			END_IF
			IF TrigNgAdd[13].Q THEN
				TodayNGClass_PM[13]:=TodayNGClass_PM[13]+1;
			END_IF
			IF TrigNgAdd[14].Q THEN
				TodayNGClass_PM[14]:=TodayNGClass_PM[14]+1;
			END_IF
			IF TrigNgAdd[15].Q THEN
				TodayNGClass_PM[15]:=TodayNGClass_PM[15]+1;
			END_IF
			IF TrigNgAdd[16].Q THEN
				TodayNGClass_PM[16]:=TodayNGClass_PM[16]+1;
			END_IF
			IF TrigNgAdd[17].Q THEN
				TodayNGClass_PM[17]:=TodayNGClass_PM[17]+1;
			END_IF
			IF TrigNgAdd[18].Q THEN
				TodayNGClass_PM[18]:=TodayNGClass_PM[18]+1;
			END_IF
			IF TrigNgAdd[19].Q THEN
				TodayNGClass_PM[19]:=TodayNGClass_PM[19]+1;
			END_IF
			IF TrigNgAdd[20].Q THEN
				TodayNGClass_PM[20]:=TodayNGClass_PM[20]+1;
			END_IF
			IF TrigNgAdd[21].Q THEN
				TodayNGClass_PM[21]:=TodayNGClass_PM[21]+1;
			END_IF
			IF TrigNgAdd[22].Q THEN
				TodayNGClass_PM[22]:=TodayNGClass_PM[22]+1;
			END_IF
			IF TrigNgAdd[23].Q THEN
				TodayNGClass_PM[23]:=TodayNGClass_PM[23]+1;
			END_IF
			IF TrigNgAdd[24].Q THEN
				TodayNGClass_PM[24]:=TodayNGClass_PM[24]+1;
			END_IF
			IF TrigNgAdd[25].Q THEN
				TodayNGClass_PM[25]:=TodayNGClass_PM[25]+1;
			END_IF
			IF TrigNgAdd[26].Q THEN
				TodayNGClass_PM[26]:=TodayNGClass_PM[26]+1;
			END_IF
			IF TrigNgAdd[27].Q THEN
				TodayNGClass_PM[27]:=TodayNGClass_PM[27]+1;
			END_IF
			IF TrigNgAdd[28].Q THEN
				TodayNGClass_PM[28]:=TodayNGClass_PM[28]+1;
			END_IF
			IF TrigNgAdd[29].Q THEN
				TodayNGClass_PM[29]:=TodayNGClass_PM[29]+1;
			END_IF
			IF TrigNgAdd[30].Q THEN
				TodayNGClass_PM[30]:=TodayNGClass_PM[30]+1;
			END_IF
		END_IF
//	END_IF
//END_FOR

(*当天夜班生产NG总数*)
TodayNG_PM:=TodayNGClass_PM[1]+TodayNGClass_PM[2]+TodayNGClass_PM[3]+TodayNGClass_PM[4]+TodayNGClass_PM[5]+
				TodayNGClass_PM[6]+TodayNGClass_PM[7]+TodayNGClass_PM[8]+TodayNGClass_PM[9]+TodayNGClass_PM[10]+
				TodayNGClass_PM[11]+TodayNGClass_PM[12]+TodayNGClass_PM[13]+TodayNGClass_PM[14]+TodayNGClass_PM[15]+
				TodayNGClass_PM[16]+TodayNGClass_PM[17]+TodayNGClass_PM[18]+TodayNGClass_PM[19]+TodayNGClass_PM[20]+
				TodayNGClass_PM[21]+TodayNGClass_PM[22]+TodayNGClass_PM[23]+TodayNGClass_PM[24]+TodayNGClass_PM[25]+
				TodayNGClass_PM[26]+TodayNGClass_PM[27]+TodayNGClass_PM[28]+TodayNGClass_PM[29]+TodayNGClass_PM[30];


	
				
CASE Data_Step OF 	
0:	
(*数据清除*)
	IF PLC_wHour=8 AND PLC_wMinute=00  AND PLC_wSecond=00 THEN
		Data_Step:=100;
	END_IF
(******清除当天数据，并记录当天日期*******)
100:
	FOR i:=1 TO 30 DO
		TodayNGClass_AM[i]:=0;(*当天白班各类NG数量*)
		TodayNGClass_PM[i]:=0;(*当天夜班各类NG数量*)
	END_FOR
	TodayNG_AM:=0;(*当天白班生产NG总数*)
	TodayNG_PM:=0;(*当天夜班生产NG总数*)
	Data_Step:=200;
200:
	SaveDataDelay(IN:=TRUE,PT:=t#2s, Q=> , ET=> );
	IF SaveDataDelay.Q THEN
		SaveDataDelay(IN:=FALSE);
		Data_Step:=0;
	END_IF
END_CASE





		
PLC_wYear;//PLC时间年
PLC_wMonth;//PLC时间月
PLC_wDay;//PLC时间日
PLC_wHour;//PLC时间时
PLC_wMinute;//PLC时间分
PLC_wSecond;//PLC时间秒

END_FUNCTION_BLOCK

// ---- POUs/BasicFunction/Data/Day_date.TcPOU
FUNCTION_BLOCK Day_date
VAR_INPUT
	dDay:INT;//实时日期；
	Hour:INT;//当前时间小时；
	Mins:INT;//分钟；
	iFinish:INT;  //尺寸检测CCD结果指示(1=完成;2=NG;3=无片;0=无效)  SizeResults
	LineScanNG:BOOL;// 极片外观判定结果   线扫NG、OK
	rTCount:BOOL;//切刀；
	Clear1: BOOL;//白班产能清零；
	Clear2: BOOL;//晚班产能清零；
	PartSelect:INT;//正负极；
	NGMark:ARRAY [0..15,0..1] OF  LREAL;//白班  0、尺寸NG；1、线扫瑕疵NG；
	NGMark2:ARRAY [0..15,0..1] OF  LREAL;//夜班  0、尺寸NG；1、线扫瑕疵NG；
	K7:REAL;//度数；
	K8: REAL;//尺寸NG类型输入1-8；
	K9:REAL;//线扫瑕疵类型输入1-8；
	EE:BOOL;
END_VAR
VAR_OUTPUT
	Cn_date:ARRAY[0..23,0..5] OF  LREAL  ;//1、裁切总数；2、瑕疵NG数；3、尺寸NG数；
	Cn_date2:ARRAY[0..10] OF  LREAL ;//白班；1、切片总数；2、线扫NG总数；3、尺寸NG总数；4、总良率；5、线扫NG率；6、尺寸NG率；
	Cn_date3:ARRAY[0..10] OF  LREAL  ;//晚班；1、切片总数；2、线扫NG总数；3、尺寸NG总数；4、总良率；5、线扫NG率；6、尺寸NG率；
END_VAR

VAR
	K1: INT;
	K2: INT;
	K3: INT;
	K4: INT;
	K5: INT;
	K6: INT;
	K11:INT;
	K12:INT;


	rRight:ARRAY [0..5] OF R_TRIG;//1、裁切一次；2、尺寸NG一次；3、线扫瑕疵NG一次；
	aTime: ARRAY [0..5] OF TON;
	AA: BOOL;
	BB: BOOL;
	CC: BOOL;
	DD:BOOL;
	FF:BOOL;

END_VAR

 K5:=REAL_TO_INT(K8);
 K6:=REAL_TO_INT(K9);

rRight[4](CLK:= FF);
 (**待机时间统计**)
IF PLC_wSecond=9 OR PLC_wSecond=19 OR PLC_wSecond=29 OR PLC_wSecond=39 OR PLC_wSecond=49 OR PLC_wSecond=59 THEN
	    FF:=TRUE;
ELSE
		FF:=FALSE;
END_IF
 
IF stSysState.iMode=1 THEN 
 	IF K7>0 AND K7<=10 THEN
		DD:=TRUE;
	ELSE
		DD:=FALSE;
	END_IF

rRight[1](CLK:=  rTCount );//裁切一次；
rRight[2](CLK:=DD AND (iFinish=2 OR  iFinish=3 ));//尺寸NG一次；
//rRight[4](CLK:=  EE AND  rTCount);//踢废吹气；
rRight[3](CLK:=DD AND (iFinish=1 OR iFinish=0)  AND K6<>8 AND K6<>0 AND NOT ProductPar.iModeEN.bCcdTcpEN AND NOT ProductPar.iModeEN.bLineScanCCDEN );//线扫NG；r
(***********切片计数***********)
IF rRight[1].Q THEN
	Cn_date[Hour,1]:=Cn_date[Hour,1]+1;
	IF Hour>=8 AND Hour<=19 THEN//白班总数；
		Cn_date2[1]:=Cn_date2[1]+1;
	END_IF
	IF Hour>=20 OR Hour<=7 THEN//晚班总数；
		Cn_date3[1]:=Cn_date3[1]+1;
	END_IF
	
END_IF
(*********瑕疵NG计数*********)
IF rRight[3].Q  AND K6<>8  AND K6<>0  THEN//IF rRight[3].Q  AND K6<>8 AND K6<>0 THEN
	Cn_date[Hour,2]:=Cn_date[Hour,2]+1;
	IF Hour>=8 AND Hour<=19 THEN//白班总数；
		Cn_date2[2]:=Cn_date2[2]+1;
	(*详细线扫NG不良统计*)	
	IF K6=1 OR K6=2 OR K6=3 OR K6=4 OR K6=5 OR K6=6 OR K6=7 OR K6=9 OR K6=10 OR K6=11 OR K6=12 OR K6=13 OR K6=14  THEN
		NGMark[K6,1]:=NGMark[K6,1]+1;
	END_IF
	END_IF
	IF Hour>=20 OR Hour<=7 THEN//晚班总数；
		Cn_date3[2]:=Cn_date3[2]+1;
	(*详细线扫NG不良统计*)	
	IF K6=1 OR K6=2 OR K6=3 OR K6=4 OR K6=5 OR K6=6 OR K6=7 OR K6=9 OR K6=10 OR K6=11 OR K6=12 OR K6=13 OR K6=14 THEN
		NGMark2[K6,1]:=NGMark2[K6,1]+1;
	END_IF
	END_IF

END_IF
(*********尺寸NG计数*********)
IF rRight[2].Q AND K5<>0 THEN
	Cn_date[Hour,3]:=Cn_date[Hour,3]+1;
	IF Hour>=8 AND Hour<=19  THEN//白班总数；
		Cn_date2[3]:=Cn_date2[3]+1;
	(*详细尺寸NG不良统计*)	
		IF K5=1 OR K5=2 OR K5=3 OR K5=4 OR K5=5 OR K5=6 OR K5=7 OR K5=8 OR K5=9 OR K5=10 OR K5=11 OR K5=12 OR K5=13 OR K5=14 THEN
			NGMark[K5,0]:=NGMark[K5,0]+1;
		END_IF
	END_IF
	IF Hour>=20 OR Hour<=7 THEN//晚班总数；
		Cn_date3[3]:=Cn_date3[3]+1;
		(*详细尺寸NG不良统计*)	
		IF K5=1 OR K5=2 OR K5=3 OR K5=4 OR K5=5 OR K5=6 OR K5=7 OR K5=8 OR K5=9 OR K5=10 OR K5=11 OR K5=12 OR K5=13 OR K5=14 THEN
			NGMark2[K5,0]:=NGMark2[K5,0]+1;
		END_IF
	END_IF

END_IF

(*自动运行时间统计*)
IF rRight[4].Q AND stSysState.iModehmi=1 THEN
	Cn_date[Hour,0]:=Cn_date[Hour,0]+1;
END_IF


(****************白班良率%*****************)
//总良率：
IF Cn_date2[1]>0 THEN
Cn_date2[4]:=(Cn_date2[1]-Cn_date2[2]-Cn_date2[3])/Cn_date2[1];
ELSE
Cn_date2[4]:=0;	
END_IF
//线扫NG率：
IF Cn_date2[1]>0 THEN
Cn_date2[5]:=Cn_date2[2]/Cn_date2[1];
ELSE
Cn_date2[5]:=0;	
END_IF
//尺寸NG率：
IF Cn_date2[1]>0 THEN
Cn_date2[6]:=Cn_date2[3]/Cn_date2[1];
ELSE
Cn_date2[6]:=0;	
END_IF

(****************晚班良率%*****************)
//总良率：
IF Cn_date3[1]>0 THEN
Cn_date3[4]:=(Cn_date3[1]-Cn_date3[2]-Cn_date3[3])/Cn_date3[1];
ELSE
Cn_date3[4]:=0;	
END_IF
//线扫NG率：
IF Cn_date3[1]>0 THEN
Cn_date3[5]:=Cn_date3[2]/Cn_date3[1];
ELSE
Cn_date3[5]:=0;	
END_IF
//尺寸NG率：
IF Cn_date3[1]>0 THEN
Cn_date3[6]:=Cn_date3[3]/Cn_date3[1];
ELSE
Cn_date3[6]:=0;	
END_IF

END_IF


(***手动时间统计**)
IF rRight[4].Q AND (stSysState.iModehmi=3 OR stSysState.iModehmi=2) THEN
	Cn_date[Hour,4]:=Cn_date[Hour,4]+1;
END_IF
/////////报警
IF rRight[4].Q AND (stSysState.iModehmi=4 OR stSysState.iModehmi=5) THEN
	Cn_date[Hour,5]:=Cn_date[Hour,5]+1;
END_IF

//白班待机时间清零
IF Clear1 OR (Hour=7 AND  Mins=20) THEN

FOR K11:=0 TO 5 DO
	 Cn_date[8,K11]:=0;
	 Cn_date[9,K11]:=0;
	 Cn_date[10,K11]:=0;
	 Cn_date[11,K11]:=0;
	 Cn_date[12,K11]:=0;
	 Cn_date[13,K11]:=0;
	 Cn_date[14,K11]:=0;
	 Cn_date[15,K11]:=0;
	 Cn_date[16,K11]:=0;
	 Cn_date[17,K11]:=0;
	 Cn_date[18,K11]:=0;
	 Cn_date[19,K11]:=0;
END_FOR
END_IF

//晚班待机时间清零
IF Clear2 OR (Hour=8 AND Mins=20 )THEN	

FOR K12:=0 TO 5 DO
	 Cn_date[20,K12]:=0;
	 Cn_date[21,K12]:=0;
	 Cn_date[22,K12]:=0;
	 Cn_date[23,K12]:=0;
	 Cn_date[0,K12]:=0;
	 Cn_date[1,K12]:=0;
	 Cn_date[2,K12]:=0;
	 Cn_date[3,K12]:=0;
	 Cn_date[4,K12]:=0;
	 Cn_date[5,K12]:=0;
	 Cn_date[6,K12]:=0;
	 Cn_date[7,K12]:=0;
END_FOR
END_IF


(***********白晚班产能清零***********)
IF Clear1 OR (Hour=7 AND  Mins=20) THEN
FOR K3:=1 TO 10 DO
	Cn_date2[K3]:=0;
END_FOR

FOR K1:=0 TO 5 DO
	 Cn_date[8,K1]:=0;
	 Cn_date[9,K1]:=0;
	 Cn_date[10,K1]:=0;
	 Cn_date[11,K1]:=0;
	 Cn_date[12,K1]:=0;
	 Cn_date[13,K1]:=0;
	 Cn_date[14,K1]:=0;
	 Cn_date[15,K1]:=0;
	 Cn_date[16,K1]:=0;
	 Cn_date[17,K1]:=0;
	 Cn_date[18,K1]:=0;
	 Cn_date[19,K1]:=0;
END_FOR
NGMark[0,0]:=0;
NGMark[1,0]:=0;
NGMark[2,0]:=0;
NGMark[3,0]:=0;
NGMark[4,0]:=0;
NGMark[5,0]:=0;
NGMark[6,0]:=0;
NGMark[7,0]:=0;
NGMark[8,0]:=0;
NGMark[9,0]:=0;
NGMark[10,0]:=0;
NGMark[11,0]:=0;
NGMark[12,0]:=0;
NGMark[13,0]:=0;
NGMark[14,0]:=0;
NGMark[0,1]:=0;
NGMark[1,1]:=0;
NGMark[2,1]:=0;
NGMark[3,1]:=0;
NGMark[4,1]:=0;
NGMark[5,1]:=0;
NGMark[6,1]:=0;
NGMark[7,1]:=0;
NGMark[8,1]:=0;
NGMark[9,1]:=0;
NGMark[10,1]:=0;
NGMark[11,1]:=0;
NGMark[12,1]:=0;
NGMark[13,1]:=0;
NGMark[14,1]:=0;
END_IF

//////////////////////////////////////////////
IF Clear2 OR (Hour=8 AND Mins=20 )THEN
FOR K4:=1 TO 10 DO
	Cn_date3[K4]:=0;
END_FOR			

